# B&R Automation Studio project x20ost
Automation Studio 3.0.71.10

## Configuration Config1

### Task classes (Cpu.sw)
```
Cyclic#4:
  bnrmain <- bnrmain.prg
DataObjects: FlashModul
Binaries: gcloader, iomap, arconfig, asfw, sysconf
Libraries: DataObj, DM_lib, sys_lib, runtime, burtrap, CAN_Lib, AsTCP, dvframe
```

### IoMap.iom - PLC1/IoMap.iom
```iecst
(********************************************************************
 * COPYRIGHT --
 ********************************************************************
 * File: IoMap.iom
 * Author: a2000
 * Created: December 09, 2009
 ********************************************************************
 * IO mapping file
 ********************************************************************)
VAR_CONFIG
	uiValueAI4_0 AT %IW.IF4.ST3.AnalogInput01;
	uiValueAI4_1 AT %IW.IF4.ST3.AnalogInput02;
	uiValueAI5_0 AT %IW.IF4.ST4.Temperature01;
	uiValueAI5_1 AT %IW.IF4.ST4.Temperature02;
	uiValueAO6_0 AT %QW.IF4.ST5.AnalogOutput01;
	uiValueAO6_1 AT %QW.IF4.ST5.AnalogOutput02;
	uiValueAO6_2 AT %QW.IF4.ST5.AnalogOutput03;
	uiValueAO6_3 AT %QW.IF4.ST5.AnalogOutput04;
	blValueDI7_0 AT %IX.IF4.ST6.DigitalInput01;
	blValueDI7_1 AT %IX.IF4.ST6.DigitalInput02;
	blValueDI7_2 AT %IX.IF4.ST6.DigitalInput03;
	blValueDI7_3 AT %IX.IF4.ST6.DigitalInput04;
	blValueDI7_4 AT %IX.IF4.ST6.DigitalInput05;
	blValueDI7_5 AT %IX.IF4.ST6.DigitalInput06;
	blValueDI7_6 AT %IX.IF4.ST6.DigitalInput07;
	blValueDI7_7 AT %IX.IF4.ST6.DigitalInput08;
	blValueDI7_8 AT %IX.IF4.ST6.DigitalInput09;
	blValueDI7_9 AT %IX.IF4.ST6.DigitalInput10;
	blValueDI7_10 AT %IX.IF4.ST6.DigitalInput11;
	blValueDI7_11 AT %IX.IF4.ST6.DigitalInput12;
	blValueDI8_0 AT %IX.IF4.ST7.DigitalInput01;
	blValueDI8_1 AT %IX.IF4.ST7.DigitalInput02;
	blValueDI8_2 AT %IX.IF4.ST7.DigitalInput03;
	blValueDI8_3 AT %IX.IF4.ST7.DigitalInput04;
	blValueDI8_4 AT %IX.IF4.ST7.DigitalInput05;
	blValueDI8_5 AT %IX.IF4.ST7.DigitalInput06;
	blValueDI8_6 AT %IX.IF4.ST7.DigitalInput07;
	blValueDI8_7 AT %IX.IF4.ST7.DigitalInput08;
	blValueDI8_8 AT %IX.IF4.ST7.DigitalInput09;
	blValueDI8_9 AT %IX.IF4.ST7.DigitalInput10;
	blValueDI8_10 AT %IX.IF4.ST7.DigitalInput11;
	blValueDI8_11 AT %IX.IF4.ST7.DigitalInput12;
	blValueDO9_0 AT %QX.IF4.ST8.DigitalOutput01;
	blValueDO9_1 AT %QX.IF4.ST8.DigitalOutput02;
	blValueDO9_2 AT %QX.IF4.ST8.DigitalOutput03;
	blValueDO9_3 AT %QX.IF4.ST8.DigitalOutput04;
	blValueDO9_4 AT %QX.IF4.ST8.DigitalOutput05;
	blValueDO9_5 AT %QX.IF4.ST8.DigitalOutput06;
	blValueDO9_6 AT %QX.IF4.ST8.DigitalOutput07;
	blValueDO9_7 AT %QX.IF4.ST8.DigitalOutput08;
	blValueDO9_8 AT %QX.IF4.ST8.DigitalOutput09;
	blValueDO9_9 AT %QX.IF4.ST8.DigitalOutput10;
	blValueDO9_10 AT %QX.IF4.ST8.DigitalOutput11;
	blValueDO9_11 AT %QX.IF4.ST8.DigitalOutput12;
	blValueDO10_0 AT %QX.IF4.ST9.DigitalOutput01;
	blValueDO10_1 AT %QX.IF4.ST9.DigitalOutput02;
	blValueDO10_2 AT %QX.IF4.ST9.DigitalOutput03;
	blValueDO10_3 AT %QX.IF4.ST9.DigitalOutput04;
	blValueDO10_4 AT %QX.IF4.ST9.DigitalOutput05;
	blValueDO10_5 AT %QX.IF4.ST9.DigitalOutput06;
	blValueDO10_6 AT %QX.IF4.ST9.DigitalOutput07;
	blValueDO10_7 AT %QX.IF4.ST9.DigitalOutput08;
	blValueDO10_8 AT %QX.IF4.ST9.DigitalOutput09;
	blValueDO10_9 AT %QX.IF4.ST9.DigitalOutput10;
	blValueDO10_10 AT %QX.IF4.ST9.DigitalOutput11;
	blValueDO10_11 AT %QX.IF4.ST9.DigitalOutput12;
END_VAR
```

## Logical view

Binary libraries used (declarations not repeated): Convert, Runtime, Operator, DataObj, DM_lib, sys_lib, CAN_Lib, AsTCP, dvframe


### Program Logical/bnrmain (ANSIC) - A new program

#### bnrmain.c - Implementation code
```c
/********************************************************************
 * COPYRIGHT -- Kontora
 ********************************************************************
 * Program: bnrmain
 * File: bnrmain.c
 * Author: Abramenya
 * Created: January 19, 2009
 ********************************************************************
 * Implementation of program bnrmain
 ********************************************************************/
#include "bnrmain.h"
#include "bnrhconfig.h"
#ifdef _DEFAULT_INCLUDES
 #include <AsDefault.h>
#endif
#ifdef WIN32
//size_t szMem;
#endif
_GLOBAL SYSxinfo_typ SYSXInfo0,SYSXInfo1;
_GLOBAL RTCtime_typ RTCGetTime, RTCSetTime;
_GLOBAL BYTE  m_byObsSystemIntState;
_GLOBAL DWORD m_dwTicTime;
CProcManager *m_pProcManager;
_GLOBAL PVOID pProcManager;
_GLOBAL PVOID pSystem;
_GLOBAL PVOID pDebMsg;
_GLOBAL DWORD nMemSize;
_GLOBAL PVOID pvMEM;
typedef struct _tagMem
{
	WORD nSize;
	void *pvMem;
}PMEM;
//_GLOBAL PMEM *m_pMEM;
extern SLMESSAGE *m_pDebMsg;
extern SHARDCOMPUTERTABLE nConfigTable;

void _INIT bnrmainINIT( void )
{
	SYSxinfo(&SYSXInfo0);
	InitSystem();
	SYSxinfo(&SYSXInfo1);
}
//Cyclic Section
_GLOBAL INT nCTT;
void _CYCLIC bnrmainCYCLIC( void )
{
	if(m_pProcManager!=0)
	m_pProcManager->Run(m_pProcManager);
	nCTT++;
	 //RTC_gettime(&RTCGetTime);
}
//Exit Section
void _EXIT bnrmainEXIT( void ){}
void InitSystem(void)
{
    InitHardValue();
    //printf("\nPre Mem");heapdump();

	m_dwTicTime = SYSTEM_QTIME;
	New(sizeof(SLMESSAGE),m_pDebMsg);

	////PMEM **m_pMEM;
	////New(sizeof(PMEM**),m_pMEM);
	////New(300*sizeof(PVOID),pvMEM);
	////pvMEM

	CreateProcManager();
	CreateSystem(&nConfigTable);
	m_pProcManager->Start(m_pProcManager);

	//pProcManager = m_pProcManager;
	//pSystem = m_pSystem;
	//pDebMsg = m_pDebMsg;
	//nMemSize = nMemSize;

	//printf("\n(__)Memory : %d",nMemSize);
	//Info("\n(__)Memory:&",&nMemSize);
	//printf("\nPost Mem");heapdump();
    //DeleteSystem();
	//nMemSize = nMemSize;
	//Status = SYSxinfo(&SYSXInfo2);
	//printf("\nPost Del Mem");heapdump();
}
void DeleteSystem(void)
{
    /*
	m_pProcManager = pProcManager;
	m_pSystem = pSystem;
	m_pDebMsg = pDebMsg;
    m_pProcManager->Stop(m_pProcManager);
	DestroyObject(CSystem,m_pSystem);
	DestroyObject(CProcManager,m_pProcManager);
	Delete(sizeof(SMESSAGE),m_pDebMsg);
	m_pProcManager = 0;
	*/
}

#ifdef WIN32
int main(void)
{
	bnrmainINIT();
	CreateCyclicProc();
	while (1)
	{
	  GetSysCommand();
	  Sleep(100);
	}
    return 0;
}
void GetSysCommand(void)
{
	int ch;
	int i=0;
	SMESSAGE sMsg;
	while((ch = getchar()) != 0x0a)
	{
	 if (i<DEV_MAX_MSG_SIZE)
	 sMsg.m_sbyInfo[1+i] = (BYTE)ch;
	 i++;
	}
	if(i>0)
	{
	 sMsg.m_sbyInfo[0]   = i+1;
     sMsg.m_swLen        = 9+i+1;
	 sMsg.m_sbyFrom      = MDL_ARMMD;
	 sMsg.m_sbyFor       = MDL_HCOMM;
	 sMsg.m_sbyIntType   = DEV_ARM_PORT_TCP;
	 sMsg.m_sbyServerID  = 0;
	 sMsg.m_sbyType      = EV_DEBMS_DEBOUT_IND;
	 sMsg.m_sbyDirection = 0xff;
	 sMsg.m_sbySensor    = 0xff;
	 //Info("\n(##)CMAIN::>HHAND:%m",(BYTE*)&sMsg);
	 FPUT(DEV_ADMIN_BOX_ID,(BYTE*)&sMsg);
	}
}
#endif
BOOL CreateProcManager(void)
{
	m_pProcManager = NULL;
	New(sizeof(CProcManager),m_pProcManager);
	InitObject(CProcManager,m_pProcManager);
	if(m_pProcManager!=NULL)
	{
	 m_pProcManager->Init(m_pProcManager,m_dwTicTime,TRUE);
 	 return TRUE;
	}else return FALSE;

}
BOOL CreateSystem(SHARDCOMPUTERTABLE *plConfigTable)
{
	m_pSystem = NULL;
	New(sizeof(CSystem),m_pSystem);
	InitObject(CSystem,m_pSystem);
	if (m_pSystem!=NULL)
	{
	 m_pSystem->CreateSystem(m_pSystem,plConfigTable);
	 return TRUE;
	}else return FALSE;
}
void DeleteTimer(PVOID pV)
{
    CSystemTimer *p;
	p = (CSystemTimer*)pV;
	m_pProcManager->DisconnectTimer(m_pProcManager,p);
}
void CrateTimer(PVOID pV)
{
    CSystemTimer *p;
	p = (CSystemTimer*)pV;
	m_pProcManager->ConnectTimer(m_pProcManager,p);
}

void CrateProcess(PVOID pV,SINT* chProcName,BYTE byStateProc,BYTE byPeriod)
{
	 CCyclicSystem *p;
	 p = (CCyclicSystem*)pV;
	 p->Create(p,chProcName,byStateProc,byPeriod);
	 m_pProcManager->ConnectProc(m_pProcManager,p);
}
_GLOBAL BYTE nYear;
void GetCurTime(STIME *pTime)
{
    #ifdef WIN32
    SYSTEMTIME nTM; WORD mSec;
	GetLocalTime(&nTM);
	pTime->tYear  = (BYTE)nTM.wYear-2000;
	pTime->tMonth = (BYTE)nTM.wMonth;
	pTime->tDay   = (BYTE)nTM.wDay;
	pTime->tHour  = (BYTE)nTM.wHour;
	pTime->tMin   = (BYTE)nTM.wMinute;

	pTime->tSec   = (BYTE)nTM.wSecond;
	mSec          = nTM.wMilliseconds + nTM.wSecond*1000;
	pTime->tMSecL = (BYTE)mSec;
	pTime->tMSecH = mSec>>8;
    #else
 	/*
      RTCSetTime.year = 2000;
      RTCSetTime.month = RTCGetTime.month;
      RTCSetTime.day = RTCGetTime.day;
      RTCSetTime.hour = RTCGetTime.hour;
      RTCSetTime.minute = RTCGetTime.minute;
      RTCSetTime.second = RTCGetTime.second;
      RTCSetTime.millisec = RTCGetTime.millisec;
      RTCSetTime.microsec = RTCGetTime.microsec;
	*/
    RTC_gettime(&RTCGetTime);
	pTime->tYear  = (RTCGetTime.year-2000);
	nYear = pTime->tYear;
	pTime->tMonth = RTCGetTime.month;
	pTime->tDay   = RTCGetTime.day;
	pTime->tHour  = RTCGetTime.hour;
	pTime->tMin   = RTCGetTime.minute;
	pTime->tSec   = RTCGetTime.second;
	RTCGetTime.millisec = RTCGetTime.millisec + ((UINT)RTCGetTime.second)*1000;
	pTime->tMSecL = (BYTE)RTCGetTime.millisec;
	pTime->tMSecH = (BYTE)(RTCGetTime.millisec>>8);
    #endif
}
void SetBoardTime(BYTE *byTime)
{
	RTCtime_typ RTCSetTime;
	BYTE nSec;
	WORD nMsec;
	RTCSetTime.year     = 2000+byTime[6];
	RTCSetTime.month    = byTime[5];
	RTCSetTime.day      = byTime[4];
	RTCSetTime.hour     = byTime[3];
	RTCSetTime.minute   = byTime[2];

	nMsec = ((WORD)byTime[0])|((WORD)byTime[1])<<8;
	nSec  = nMsec/1000;
    nMsec = nMsec - nSec*1000;

	RTCSetTime.second   = nSec;
	RTCSetTime.millisec = nMsec;
	//Info("\nYR:%w MN:%b DY:%b HR:%b MI:%b SC:%b MS:%w",&RTCSetTime.year,&RTCSetTime.month,&RTCSetTime.day,&RTCSetTime.hour,&RTCSetTime.minute,&nSec,&nMsec);
    #ifndef WIN32
	RTC_settime(&RTCSetTime);
    #endif
}
void SendSMessage(BYTE byBox,BYTE byFor,BYTE byType)
{
    SHORTMESSAGE m_sMsg;
	m_sMsg.m_swLen        = 9;
	m_sMsg.m_sbyFrom      = DIR_PHMDL;
	m_sMsg.m_sbyFor       = byFor;
	m_sMsg.m_sbyIntType   = 0;
	m_sMsg.m_sbyServerID  = 0;
	m_sMsg.m_sbyType      = byType;
	m_sMsg.m_sbyDirection = 0;
	m_sMsg.m_sbySensor    = 0;
	FPUT(byBox,(BYTE*)&m_sMsg);
    #ifdef DEB_CMain
	Info("\n(__)CMAIN::>OUTT::%M",&m_sMsg);
    #endif
}
void SendCommand(BYTE byEvent,SINT *pchCommand)
{
	SHORTMESSAGE m_sMsg;
	BYTE byNbLen;
	m_sMsg.m_sbyFrom      = DIR_KPMOD;
	m_sMsg.m_sbyFor       = DIR_KPTO101;
	m_sMsg.m_sbyIntType   = 0;
	m_sMsg.m_sbyServerID  = 0;
	m_sMsg.m_sbyType      = byEvent;
	m_sMsg.m_sbyDirection = 0;
	m_sMsg.m_sbySensor    = 0;
	byNbLen = strlen(pchCommand);
    memcpy(m_sMsg.m_sbyInfo,pchCommand,byNbLen);
	m_sMsg.m_sbyInfo[byNbLen] = 13;
	m_sMsg.m_sbyInfo[byNbLen+1] = 10;
	m_sMsg.m_swLen            = 9+byNbLen+2;
	#ifdef DEB_CMain
    Info("\n(__)CMAIN::>Command:%s",pchCommand);
    #endif
	FPUT(DEV_RSMMD_BOX_ID,(BYTE*)&m_sMsg);
}
void SendChar(BYTE byEvent,SINT *pchCommand)
{
	SHORTMESSAGE m_sMsg;
	BYTE byNbLen;
	m_sMsg.m_sbyFrom      = DIR_KPMOD;
	m_sMsg.m_sbyFor       = DIR_KPTO101;
	m_sMsg.m_sbyIntType   = 0;
	m_sMsg.m_sbyServerID  = 0;
	m_sMsg.m_sbyType      = byEvent;
	m_sMsg.m_sbyDirection = 0;
	m_sMsg.m_sbySensor    = 0;
	byNbLen = strlen(pchCommand);
    memcpy(m_sMsg.m_sbyInfo,pchCommand,byNbLen);
	//m_sMsg.m_sbyInfo[byNbLen] = 13;
	//m_sMsg.m_sbyInfo[byNbLen+1] = 10;
	m_sMsg.m_swLen            = 9+byNbLen;
	//#ifdef DEB_CMain
    //Info("\n(__)CMAIN::>Command:%s",pchCommand);
    //#endif
	FPUT(DEV_RSMMD_BOX_ID,(BYTE*)&m_sMsg);
}
_GLOBAL INT nQMem;
void NEW(int nSize,void **pVoid)
{
     #ifdef WIN32
	 MEM_alloc(nSize,*pVoid);
     #else
	 MEM_alloc(nSize,pVoid);
     #endif
	 nQMem++;
	 nMemSize += nSize;
};
void FREE(int nSize,void **pVoid)
{
	 if(nSize!=0)
     MEM_free(nSize,pVoid);
	 nMemSize -= nSize;
}
#ifdef WIN32
DWORD WINAPI CyclicProcess( PVOID pVoid)
{
	HANDLE hEvent = CreateEvent(NULL,FALSE,TRUE,NULL);
	int nTime;
	while (1)
	{
	 bnrmainCYCLIC();
	 WaitForSingleObject(hEvent,m_dwTicTime);
	 //if (nTime%50==0) Info("\nTMR_________");
	 //nTime++;
	 //Sleep(20);
	 //Sleep(m_dwTicTime);
	}
	return 0;
}
void CreateCyclicProc(void)
{
	DWORD dwThreadId, dwThrdParam = 1;
	HANDLE hThread;
	hThread = CreateThread(NULL,0,CyclicProcess,&dwThrdParam,0,&dwThreadId);
}
void heapdump( void )
{
	_HEAPINFO hinfo;
	int heapstatus;
	hinfo._pentry = NULL;
	while( ( heapstatus = _heapwalk( &hinfo ) ) == _HEAPOK )
	{ printf( "%6s block at %Fp of size %4.4X\n",
	( hinfo._useflag == _USEDENTRY ? "USED" : "FREE" ),
	hinfo._pentry, hinfo._size );
	}

	switch( heapstatus )
	{
	case _HEAPEMPTY:
		printf( "OK - empty heap\n" );
		break;
	case _HEAPEND:
		printf( "OK - end of heap\n" );
		break;
	case _HEAPBADPTR:
		printf( "ERROR - bad pointer to heap\n" );
		break;
	case _HEAPBADBEGIN:
		printf( "ERROR - bad start of heap\n" );
		break;
	case _HEAPBADNODE:
		printf( "ERROR - bad node in heap\n" );
		break;
	}
}
#endif
```

#### bnradmin.c
```c
/********************************************************************
 * COPYRIGHT -- Kontora
 ********************************************************************
 * Program: bnrmain
 * File: bnrlsens.c
 * Author: Abramenya
 * Created: January 19, 2009
 *******************************************************************/

#include "bnradmin.h"
#include "bnrpob.h"
#ifdef _DEFAULT_INCLUDES
 #include <AsDefault.h>
#endif
#define SYS_REQ_ALL_PARAM                0x6673 // isf - Авария интерфейса
#define SYS_SET_OUT                      0x746f // iot xxx
#define SYS_SET_OUT_BOX                  0x626f // iob xxx
#define SYS_SET_TST_MSG                  0x6d74 // itm xxx
#define SYS_SET_OUT_DIR                  0x736f // iob xxx
#define SYS_SET_DEV_VER                  0x766f // iov xxx
extern SSOFTSWITCHTABLE nSoftSwitchTable;
extern BOOL *blpValueDI8[];
extern UINT *uipValueAI2[];

extern BOOL *blpAlValueAI2[];
extern BOOL *blAsValueAI[];
//_GLOBAL INT iCAdminVal;
SINT *chAdmState[] =
{
	"ST00_NULL",
    "ST01_DISC",
	"ST02_CONN",
	"ST03_WAIT_CONF",
	"ST04_SYST_READY",
	"ST05_WAIT_READY",
};
_GLOBAL INT16 wTICode,nSG;
void CAdmin_Init(This)
{
     DECLARE_MULTI_OPEN(CAdmin,CCyclicSystem)
     #ifdef DEB_CAdmin
	 Info("\n(__)CADMN::>Create Admin.");
     #endif
	 wTICode = 0;
	 nSG     = 0;
	 //pT->m_blArmState = FALSE;
	 //dwFL  |= DEB_OUT_BOX_ADMIN;
	 //dwFL = 48;
	 pB->SetBoxID(pB,DEV_ADMIN_BOX_ID);
	 pT->m_bySystemState = SYS_ST01_DISC;
	 pT->m_blArmState = TRUE;
}
_GLOBAL UINT nTICHA;
void CAdmin_CyclicProc(This)
{
     DECLARE_MULTI_OPEN(CAdmin,CCyclicSystem)
	 pB->m_dwAmoutQuant++;

	 if(wTICode>=32000)
	 nSG = -400;
	 if(wTICode<=0)
	 nSG = 400;

	 //wTICode =  wTICode + nSG;
	 //*uipValueAI2[0] = wTICode;

	 //nTICHA++;
	 //if ((nTICHA % 2)==0)
	 //Info("\n(__)CADMN::>TI:%w",uipValueAI2[0]);
}

void CAdmin_SetSystemID(This,BYTE bySystemID)
{
     DECLARE_MULTI_OPEN(CAdmin,CCyclicSystem)
	 pT->m_bySystemID = bySystemID;
}
BOOL CAdmin_EventHandler(This,SMESSAGE *pMsg)
{
	 BOOL res = TRUE;
     DECLARE_MULTI_OPEN(CAdmin,CCyclicSystem)
	 BYTE byState;
	 byState = pT->GetState(pT);
	 switch (pMsg->m_sbyFor)
	 {
		case MDL_HCOMM:
			 pT->PreCommHandler(pT,pMsg);
		break;
		case MDL_ADMIN:
			 pT->AdminAutomat(pT,pMsg);
		break;
		case MDL_SYSTM:
		break;
		case MDL_DIRMD:
		break;
		case MDL_COMPT:
		break;
		default:
		break;
	 }
	 return res;
}
BOOL CAdmin_AdminAutomat(This,SMESSAGE *pMsg)
{
     DECLARE_MULTI_OPEN(CAdmin,CCyclicSystem)
	 BOOL res = FALSE;
	 BYTE byEvent = pMsg->m_sbyType;
	 switch(pT->GetState(pT))
	 {
	    case SYS_ST00_NULL:
        break;
	    case SYS_ST01_DISC:
			 if((byEvent==EV_ADMIN_ARM_CONN_IND))
			 {
              #ifdef DEB_CAdmin
			  Info("\n(%b)CADMN::>ARM_CONN_IND:%M",&pT->m_bySystemID,(BYTE*)pMsg);
              #endif
			  pT->m_blArmState = TRUE;
              pT->SendMessage(pT,DEV_ARMOT_BOX_ID,MDL_ARMSY,EV_ADMIN_ARM_CONN_IND,0,0);
			  pT->SendMessage(pT,DEV_ARMOT_BOX_ID,MDL_ARMSY,EV_ADMIN_SYS_CONFIG_IND,0,0); //Запросить конфигурацию
			  pT->m_pTAskConfig.OnTimer(&pT->m_pTAskConfig,T4SEC);
			  pT->SetState(pT,SYS_ST03_WAIT_CONF);
			  res = TRUE;
			 }
        break;
		case SYS_ST02_CONN:
        break;
	    case SYS_ST03_WAIT_CONF:
			 if(byEvent==EV_ADMIN_ASK_CONF_TIM_IND)
			 {
              #ifdef DEB_CAdmin
			  Info("\n(%b)CADMN::>ASK_CONF_TIM_IND:%M",&pT->m_bySystemID,(BYTE*)pMsg);
              #endif
			  pT->SendMessage(pT,DEV_ARMOT_BOX_ID,MDL_ARMSY,EV_ADMIN_SYS_CONFIG_IND,0,0); //Запросить конфигурацию
			  pT->m_pTAskConfig.OnTimer(&pT->m_pTAskConfig,T4SEC);
			  res = TRUE;
			 }else
			 if(byEvent==EV_ADMIN_SYS_CONFIG_REQ)
			 {
              #ifdef DEB_CAdmin
			  Info("\n(%b)CADMN::>SYS_CONFIG_REQ:%M",&pT->m_bySystemID,(BYTE*)pMsg);
              #endif
			  pT->m_pTAskConfig.OfTimer(&pT->m_pTAskConfig);
			  pT->SendMessage(pT,DEV_SYSTM_BOX_ID,MDL_SYSTM,EV_SYSTM_INIT_OBS_REQ,0,0);
			  res = TRUE;
			 }else
			 if(byEvent==EV_SYSTM_INIT_OBS_IND)
			 {
              #ifdef DEB_CAdmin
			  Info("\n(%b)CADMN::>INIT_OBS_IND:%M",&pT->m_bySystemID,(BYTE*)pMsg);
              #endif
			  Info("\n(%b)CADMN::>B&R System Ready!",&pT->m_bySystemID);
			  pT->SendMessage(pT,DEV_ARMOT_BOX_ID,MDL_ARMSY,EV_ADMIN_SYS_READY_IND,0,0);
			  pT->SetState(pT,SYS_ST04_SYST_READY);
			  res = TRUE;
			 }
			 if(byEvent==EV_ADMIN_ARM_DISC_IND)pT->SetState(pT,SYS_ST01_DISC);
        break;
		case SYS_ST05_WAIT_READY:
			 switch(byEvent)
			 {
			  case EV_ADMIN_TMR_SSTATE_IND:
				   pT->SendMessage(pT,DEV_ARMOT_BOX_ID,MDL_ARMSY,EV_ADMIN_SYS_READY_IND,0,0);
				   pT->m_pTSendState.OnTimer(&pT->m_pTSendState,T4SEC);
			  break;
			  case EV_ADMIN_ARM_READY_REQ:
				   //pT->m_pTSendState->OfTimer(pT->m_pTSendState);
				   pT->SendMessage(pT,DEV_ARMOT_BOX_ID,MDL_ARMSY,EV_ADMIN_SYS_READY_IND,0,0);
				   pT->m_blArmState = TRUE;
				   pT->SetState(pT,SYS_ST04_SYST_READY);
			  break;
			  default:
			  break;
			 }
		break;
	    case SYS_ST04_SYST_READY:
			 switch(byEvent)
			 {
			  case EV_ADMIN_ARM_READY_REQ:
				   pT->SendMessage(pT,DEV_ARMOT_BOX_ID,MDL_ARMSY,EV_ADMIN_SYS_READY_IND,0,0);
			  break;
			  case EV_ADMIN_ARM_DISC_IND:
				   //pT->m_pTSendState->OnTimer(pT->m_pTSendState,T4SEC);
				   pT->SetState(pT,SYS_ST05_WAIT_READY);
				   pT->m_blArmState = FALSE;
			  break;
			  case EV_ADMIN_SET_ALM_HILEV_REQ: //Авария превышения верхнего ав. предела 	68
                   #ifdef DEB_CAdmin
			       Info("\n(%b)CADMN::>SET_ALM_HILEV_REQ:%M",&pT->m_bySystemID,(BYTE*)pMsg);
                   #endif
			   	   pT->SendMessage(pT,DEV_ARMOT_BOX_ID,MDL_ARMSY,pMsg->m_sbyType,pMsg->m_sbyDirection,pMsg->m_sbySensor);
			  break;
			  case EV_ADMIN_REM_ALM_HILEV_REQ: //Устранение аварии превышения верхнего ав. предела 	69
                   #ifdef DEB_CAdmin
			       Info("\n(%b)CADMN::>REM_ALM_HILEV_REQ:%M",&pT->m_bySystemID,(BYTE*)pMsg);
                   #endif
			       pT->SendMessage(pT,DEV_ARMOT_BOX_ID,MDL_ARMSY,pMsg->m_sbyType,pMsg->m_sbyDirection,pMsg->m_sbySensor);
			  break;
			  case EV_ADMIN_SET_ALM_LOLEV_REQ: //Авария превышения нижнего ав. предела 	70
                   #ifdef DEB_CAdmin
			       Info("\n(%b)CADMN::>REM_ALM_LOLEV_REQ:%M",&pT->m_bySystemID,(BYTE*)pMsg);
                   #endif
			       pT->SendMessage(pT,DEV_ARMOT_BOX_ID,MDL_ARMSY,pMsg->m_sbyType,pMsg->m_sbyDirection,pMsg->m_sbySensor);
			  break;
			  case EV_ADMIN_REM_ALM_LOLEV_REQ: //Устранение аварии превышения нижнего ав. предела 	71
                   #ifdef DEB_CAdmin
			       Info("\n(%b)CADMN::>REM_ALM_LOLEV_REQ:%M",&pT->m_bySystemID,(BYTE*)pMsg);
                   #endif
			       pT->SendMessage(pT,DEV_ARMOT_BOX_ID,MDL_ARMSY,pMsg->m_sbyType,pMsg->m_sbyDirection,pMsg->m_sbySensor);
			  break;
	          case EV_ADMIN_ARM_STOP_REQ:
		           //pT->CloseInterface(pC);
			       //Info("\n(%b)CADMN::>EV_ADMIN_ARM_STOP_REQ:%M",&pT->m_bySystemID,(BYTE*)pMsg);
	       	  break;
			 }
        default:
		break;
	 }
	 return res;
}
BOOL CAdmin_SendMessage(This,BYTE byBox,BYTE byFor,BYTE byType,BYTE byDir,BYTE bySens)
{
     DECLARE_MULTI_OPEN(CAdmin,CCyclicSystem)
	 BOOL res = TRUE;
	 SHORTMESSAGE m_sMsg;
	 m_sMsg.m_swLen        = 9;
	 m_sMsg.m_sbyFrom      = MDL_ADMIN;
	 m_sMsg.m_sbyFor       = byFor;
	 m_sMsg.m_sbyIntType   = DEV_SYS_INTERFACE;
	 m_sMsg.m_sbyServerID  = pT->m_bySystemID;
	 m_sMsg.m_sbyType      = byType;
	 m_sMsg.m_sbyDirection = byDir;
	 m_sMsg.m_sbySensor    = bySens;
	 //if(pT->m_blArmState)
     FPUT(byBox,(BYTE*)&m_sMsg);
	 return res;
}
void CAdmin_PreCommHandler(This,SMESSAGE *pMsg)
{
     DECLARE_MULTI_OPEN(CAdmin,CCyclicSystem)
	 BYTE byLength;
	 DWORD Code;
	 BYTE ps,*pD=(BYTE*)&Code;
     #ifdef DEB_CAdmin
 	 Info("\n(__)CHAND::>HSYST_O <- %m",pMsg->m_sbyInfo);
     #endif
	 Code = 0;
	 byLength = pMsg->m_sbyInfo[0];
	 for (ps = 0;ps<byLength;ps++)
	 if ((char)pMsg->m_sbyInfo[ps]==' ')
	 break;
	 if (ps<=MAX_COMMAND_LENGTH)
	 {
	 #ifdef WIN32
	 memcpy(&Code,&pMsg->m_sbyInfo[2],ps-2);
	 #else
	 pD[3] = pMsg->m_sbyInfo[2];
	 pD[2] = pMsg->m_sbyInfo[3];
	 #endif
	 pT->HandCommHandler(pT,Code,ps,pMsg->m_sbyInfo,byLength);

	 }
}
void CAdmin_HandCommHandler(This,DWORD b_lCode,BYTE ps,BYTE *pbyBuffer,BYTE byLength)
{
     DECLARE_MULTI_OPEN(CAdmin,CCyclicSystem)
	 SHORTMESSAGE m_sMsg;
	 BYTE byParam0,byParam1;
	 WORD wValue;
	 #ifdef DEB_CAdmin
	 //Info("\n(##)CHAND::>Code:%d, PS:%b LN:%b MS0:%b",&b_lCode,&ps,&byLength,&pbyBuffer[ps]);
     #endif
	 switch(b_lCode)
	 {
       case SYS_REQ_ALL_PARAM:
		   if (ps<(byLength-1))
		   {
            ps++;
			byParam0=pbyBuffer[ps]-0x30;
		    //Info("\nCHAND::>Command SYS_REQ_ALL_PARAM.Param0:%b",&byParam0);
		   }
	   break;
       case SYS_SET_TST_MSG:// itm xxx
		    if (ps<(byLength-1))
			{
			   ps++;
			   byParam0=pbyBuffer[ps]-0x30;
			   ps++;
			   byParam1=pbyBuffer[ps]-0x30;
               #ifdef DEB_CAdmin
			   Info("\n(__)CHAND::>SET DIG PIN[%b]:STT[%b]",&byParam0,&byParam1);
			   #endif
			   *blpValueDI8[byParam0] = byParam1;
			   //*blpAlValueAI2[byParam0] = byParam1;
			   //*blAsValueAI = byParam1;
			   //Info("\n(%b)SetPin In %b",&byParam0,&byParam1);
			}
	   break;
       case SYS_SET_OUT://iot
		   {
		    ps++;
		    if((pbyBuffer[ps]-0x30)) dwFL |= DEB_OUT_CYC_ADMIN;else dwFL &= ~DEB_OUT_CYC_ADMIN;
		    ps++;
		    if((pbyBuffer[ps]-0x30)) dwFL |= DEB_OUT_CYC_SYSTM;else dwFL &= ~DEB_OUT_CYC_SYSTM;
		    ps++;
		    if((pbyBuffer[ps]-0x30)) dwFL |= DEB_OUT_CYC_OBSRV;else dwFL &= ~DEB_OUT_CYC_OBSRV;
			ps++;
			if((pbyBuffer[ps]-0x30)) dwFL |= DEB_OUT_PMAN_STAT;else dwFL &= ~DEB_OUT_PMAN_STAT;
		    Info("\n(__)CHAND::>Out SYS_SET_OUT[%w] ",&dwFL);
		   }
       break;
       case SYS_SET_OUT_DIR://ios
		   {
		    ps++;
		    if((pbyBuffer[ps]-0x30)) dwFL |= DEB_OUT_OBSR_COMM;else dwFL &= ~DEB_OUT_OBSR_COMM;
		    ps++;
		    if((pbyBuffer[ps]-0x30)) dwFL |= DEB_OUT_DIRC_COMM;else dwFL &= ~DEB_OUT_DIRC_COMM;
		    Info("\n(__)CHAND::>Out SYS_SET_OUT_DIR[%w] ",&dwFL);
		   }
       break;
	   case SYS_SET_OUT_BOX: //iob
		   {
			ps++;
			if((pbyBuffer[ps]-0x30)) dwFL |= DEB_OUT_BOX_ADMIN;else dwFL &= ~DEB_OUT_BOX_ADMIN;
			ps++;
			if((pbyBuffer[ps]-0x30)) dwFL |= DEB_OUT_BOX_SYSTM;else dwFL &= ~DEB_OUT_BOX_SYSTM;
			ps++;
			if((pbyBuffer[ps]-0x30)) dwFL |= DEB_OUT_BOX_OBSRV;else dwFL &= ~DEB_OUT_BOX_OBSRV;
			Info("\n(__)CHAND::>Out SYS_SET_OUT_[%w]",&dwFL);
		   }
	   break;
	   case SYS_SET_DEV_VER:// iov
           pT->DevVersion(pT) ;
	   break;
	   default:
	   break;
	 };
}
void CAdmin_DevVersion(This)
{
	  DECLARE_MULTI_OPEN(CAdmin,CCyclicSystem)
	  Info("\n/----------------/Automation 2k/---------------------------/");
	  Info("\n/ Объект     :Бобруйский ЗСКГШ............................./");
      #if MYSYSTEM_ID==0
	  Info("\n/ Назначение :Управление параметрами в контуре АС-1......../");
      #elif MYSYSTEM_ID == 1
	  Info("\n/ Назначение :Управление параметрами в контуре АС-2......../");
	  #elif MYSYSTEM_ID == 2
	  Info("\n/ Назначение :Управление параметрами в контуре АС-3......../");
      #elif MYSYSTEM_ID == 3
	  Info("\n/ Назначение :Управление параметрами в контуре КОП........./");
      #elif MYSYSTEM_ID == 4
	  Info("\n/ Назначение :Управление ЧРЭП............................../");
	  #endif
	  Info("\n/ Версия     :[09.09.2009]................................./");
	  Info("\n/ Устройство :Контроллер B&R 2005........................../");
	  Info("\n/ Разработчик:Абраменя Александр Васильевич(2009г)........./");
	  Info("\n/ Тел/mail   :(8-029-563-76-78/alex_mpowt@tut.by)........../");
	  Info("\n/----------------------------------------------------------/");
}
void CAdmin_SetState(This,BYTE byState)
{
     DECLARE_MULTI_OPEN(CAdmin,CCyclicSystem)
     #ifdef DEB_CAdmin
	 Info("\n(%b)CADMN::>State:(%s)->(%s):",&pT->m_bySystemID,chAdmState[pT->m_bySystemState],chAdmState[byState]);
     #endif
     pT->m_bySystemState = byState;
}
BYTE CAdmin_GetState(This)
{
     DECLARE_MULTI_OPEN(CAdmin,CCyclicSystem)
	 return pT->m_bySystemState;
}
void CAdmin_CAdmin(This)
{
     DECLARE_MULTI_OPEN(CAdmin,CCyclicSystem)
	 DECLARE_REGISTRATION(CAdmin,Init)
	 DECLARE_REGISTRATION(CAdmin,SendMessage)
	 DECLARE_REGISTRATION(CAdmin,HandCommHandler)
	 DECLARE_REGISTRATION(CAdmin,PreCommHandler)
	 DECLARE_REGISTRATION(CAdmin,SetSystemID)
	 DECLARE_REGISTRATION(CAdmin,SetState)
	 DECLARE_REGISTRATION(CAdmin,GetState)
	 DECLARE_REGISTRATION(CAdmin,AdminAutomat)
	 DECLARE_REGISTRATION(CAdmin,DevVersion)
	 DECLARE_VIRTUAL_FUNC(CAdmin,CyclicProc)
	 DECLARE_VIRTUAL_FUNC(CAdmin,EventHandler)
	 InitObject(CMTimer,&pT->m_pTAskConfig);
     pT->m_pTAskConfig.SetTimer(&pT->m_pTAskConfig,MDL_ADMIN,MDL_ADMIN,EV_ADMIN_ASK_CONF_TIM_IND,0,0,DEV_ADMIN_BOX_ID);
	 InitObject(CMTimer,&pT->m_pTSendState);
     pT->m_pTSendState.SetTimer(&pT->m_pTSendState,MDL_ADMIN,MDL_ADMIN,EV_ADMIN_TMR_SSTATE_IND,0,0,DEV_ADMIN_BOX_ID);
}
void CAdmin_DCAdmin(This)
{
	 DECLARE_MULTI_OPEN(CAdmin,CCyclicSystem)
}
DECLARE_MULTI_CREATE(CAdmin,CCyclicSystem)
```

#### bnrkp.c
```c
/********************************************************************
 * COPYRIGHT -- Kontora
 ********************************************************************
 * Program: bnrmain
 * File: bnrlsens.c
 * Author: Abramenya
 * Created: January 19, 2009
 *******************************************************************/

#include "bnrkp.h"
#include "bnrmain.h"
#ifdef _DEFAULT_INCLUDES
 #include <AsDefault.h>
#endif
extern SKPPARAM nKP;
extern SARMINTERFACE nARM0;
extern STIPARAMS nTI;
extern STSPARAMS nTS;
extern STUPARAMS nTU;
extern char *STTS[];
_GLOBAL INT nSendTmrQry;
void CKpModule_Init(This,SHARDCOMPUTERTABLE *pPCTable,SSOFTSWITCHTABLE *pKPTable)
{
    DECLARE_MULTI_OPEN(CKpModule,CCyclicSystem)
	BOOL blSerialize;
	//pT->m_byKpID = pKPTable->sDirectionTable[0].byDirectionID;
	FDEFINE(DEV_KPMDL_BOX_ID,DEV_KPMDL_BOX_SZ);
    FDEFINE(BOX_L4,BOX_L4_SZ);
	FDEFINE(BOX_L4_1,BOX_L4_1_SZ);
	nSendTmrQry = 0;
    InitObject(CMFlash,&pT->m_nFlash);
	pT->m_pFlash = &pT->m_nFlash;
    pB->SetBoxID(pB,DEV_KPMDL_BOX_ID);
	pT->m_pPCT   = pPCTable;
	pT->m_pPST   = pKPTable;
	pT->m_pKP    = pPCTable->pKpParam;
	pT->m_byKpID = pT->m_pKP->byKpID;
	pT->m_pD     = &pT->m_pPST->sDirectionTable[0];
	pT->m_wCallTime = pT->m_pKP->byCallPeriod*10;
	pT->m_blDiscStart = FALSE;
	pT->m_byDiscProc  = 0;

	pT->m_byObsObject = 0;
	pT->m_byObsTime   = 0;
	pT->m_blIfConnect = TRUE;

    pT->m_byKpState    = MKP_NULL_ST00;
	//pT->m_byConnCT = 0;
	pT->m_blBufferST = TRUE;
	InitObject(CMTimer,&pT->m_nConnTMR);
	pT->m_nConnTMR.SetTimer(&pT->m_nConnTMR,DIR_KPTOKP,DIR_KPTOKP,EV_TMR_SRR_REQ,0,0,DEV_KPMDL_BOX_ID);

	InitObject(CMTimer,&pT->m_nRepConnTMR);
	pT->m_nRepConnTMR.SetTimer(&pT->m_nRepConnTMR,DIR_KPTOKP,DIR_KPTOKP,EV_TMR_RCAL_REQ,0,0,DEV_KPMDL_BOX_ID);

	InitObject(CMTimer,&pT->m_nDiscTMR);
	pT->m_nDiscTMR.SetTimer(&pT->m_nDiscTMR,DIR_KPTOKP,DIR_KPTOKP,EV_TMR_DISC_REQ,0,0,DEV_KPMDL_BOX_ID);

	InitObject(CMTimer,&pT->m_pResetTimer);
 	pT->m_pResetTimer.SetTimer(&pT->m_pResetTimer,DIR_KPTOKP,DIR_KPTOKP,EV_SYSTM_RESET_TIM_BRD_IND,0,0,DEV_KPMDL_BOX_ID);

	InitObject(CMTimer,&pT->m_nConnRepTMP);
	pT->m_nConnRepTMP.SetTimer(&pT->m_nConnRepTMP,DIR_KPTOKP,DIR_KPTOKP,EV_TMR_CNRP_REQ,0,0,DEV_KPMDL_BOX_ID);

	InitObject(CMTimer,&pT->m_nPuCommTMR);
	pT->m_nPuCommTMR.SetTimer(&pT->m_nPuCommTMR,DIR_KPTOKP,DIR_KPTOKP,EV_TMR_PUCM_REQ,0,0,DEV_KPMDL_BOX_ID);

	InitObject(CMTimer,&pT->m_nSDiscTMR);
	pT->m_nSDiscTMR.SetTimer(&pT->m_nSDiscTMR,DIR_KPTOKP,DIR_KPTOKP,EV_TMR_SDIS_REQ,0,0,DEV_KPMDL_BOX_ID);

	blSerialize = pT->Serialize(pT,FALSE);
	pT->CreateChannels(pT,&pKPTable->sDirectionTable[0]);

	#ifdef DEB_CKpModule
 	Info("\n(__)CKPMD::>Create Kp Module");
    #endif
	//pT->SaveInPin(pT);
}
_GLOBAL BYTE nTUU;
void CKpModule_CreateChannels(This,SDIRTABLE *pDTable)
{
    DECLARE_MULTI_OPEN(CKpModule,CCyclicSystem)
	WORD i;
	CTeleInd *pTI;
	CTeleSignal *pTS;
	CTeleControl *pTU;
	STSPARAM *pPV;
	pT->m_wAmChannel = pDTable->byAmSwitching;
	New(sizeof(CTeleSensor*)*pT->m_wAmChannel,pT->m_pTeleSensor);
	for(i=0;i<pT->m_wAmChannel;i++)
	{
	 pPV = (STSPARAM*)pDTable->pSwitchTable[i];//Find Type
	 switch (pPV->byType)
	 {
	   case TI:
		    New(sizeof(CTeleInd),pTI);
			InitObject(CTeleInd,pTI);
			pTI->pBase->m_pComputer = pT->m_pComputer;
			pT->m_pTeleSensor[i]    = pTI->pBase;
			pTI->pBase->m_pPCT      = pT->m_pPCT;
			pTI->pBase->Init(pTI->pBase,(PVOID)pPV);
	   break;
	   case TS:
		    New(sizeof(CTeleSignal),pTS);
			InitObject(CTeleSignal,pTS);
			pTS->pBase->m_pComputer = pT->m_pComputer;
		    pT->m_pTeleSensor[i]    = pTS->pBase;
			pTS->pBase->m_pPCT      = pT->m_pPCT;
			pTS->pBase->Init(pTS->pBase,(PVOID)pPV);
	   break;
	   case TU:
		    New(sizeof(CTeleControl),pTU);
			InitObject(CTeleControl,pTU);
			pTU->pBase->m_pComputer = pT->m_pComputer;
		    pT->m_pTeleSensor[i]    = pTU->pBase;
			pTU->pBase->m_pPCT      = pT->m_pPCT;
			pTU->pBase->Init(pTU->pBase,(PVOID)pPV);
	   break;
	   default:
	   break;
	 }
	}
}
/*
REG_KPPAR_ADDR=0,
REG_PORTT_ADDR,
REG_HARDT_ADDR,
REG_SOFTI_ADDR,
REG_SOFTS_ADDR,
REG_SOFTU_ADDR,
REG_SOFTR_ADDR,
*/
BOOL CKpModule_EventHandler(This,SMESSAGE *pMsg)
{
    DECLARE_MULTI_OPEN(CKpModule,CCyclicSystem)
	CTeleSensor *pTS;
	WORD wValue = 0;
	BYTE byID;
	BYTE byA0   = pMsg->m_sbyInfo[1];
	BYTE byA1   = pMsg->m_sbyInfo[2];
	BYTE byA2   = pMsg->m_sbyInfo[3];
	BYTE byLen  = pMsg->m_sbyInfo[0];
	WORD wParam;
	#ifdef DEB_CKpModule
	Info("\n(__)CKPMM::>INPT::%M",pMsg);
	#endif
	switch(pMsg->m_sbyFor)
	{
	  case DIR_101TOKP:
		   switch(pMsg->m_sbyType)
		   {
		    case PL_DATA_IND:
				 switch(byA0)
				 {
				   case REG_KPPAR_ADDR:
					    if ((byA1 == CKP_SETT_TIME)||(byA1 == CKP_SETT_KPID))
						{
						    if (byA1 == CKP_SETT_TIME) SetBoardTime(&pMsg->m_sbyInfo[4]);
							pT->m_nPuCommTMR.OfTimer(&pT->m_nPuCommTMR);
							pT->m_nConnTMR.OfTimer(&pT->m_nConnTMR);
							pT->m_nConnRepTMP.OfTimer(&pT->m_nConnRepTMP);
							//pT->m_nRepConnTMR.OfTimer(&pT->m_nRepConnTMR);
							//pT->m_blIfConnect = FALSE;
							#ifdef DEB_CKpModule
	    					Info("\n(__)CKPMM::>PU TIMER OFF");
							#endif
						}
				   	    if (byA1 == CKP_CLSE_PORT) SendSMessage(DEV_RSMMD_BOX_ID,DIR_KPTOPH,PH_CLOSE_PORT_REQ);
						if (byA1 == CKP_SAVE_SETT) {pT->m_nCT.byDefSett = 0;pT->Serialize(pT,TRUE);}
						if (byA1 == CKP_REST_BORD) pT->m_pResetTimer.OnTimer(&pT->m_pResetTimer,100);
						if (byA1 == CKP_REST_12BR)
						{
						 memcpy(&wParam,&pMsg->m_sbyInfo[5],2);
						 pT->m_nCT.byDefSett = (BYTE)wParam;
				         pT->Serialize(pT,TRUE);
						 pT->m_pResetTimer.OnTimer(&pT->m_pResetTimer,100);
						}
						if (byA1 == CKP_STOP_REST) pT->m_pResetTimer.OfTimer(&pT->m_pResetTimer);
						if (byA1 == CKP_FREE_BXL4) FFREE(BOX_L4);
						if (byA1 == CKP_SETT_BL41) pT->SaveInPin(pT);
						if (byA1 == CKP_REMT_DISC) pT->m_nSDiscTMR.OnTimer(&pT->m_nSDiscTMR,30);
						if (byA1 == CKP_SVAL_PINS) pT->SaveAlarmPin(pT);
						if (byA1 == CKP_SVAL_SLOT) pT->SaveSlotState(pT);
						if (byA1 == CKP_STRT_CHTM)
						{
							#ifdef WIN32
							pT->m_byObsObject = pMsg->m_sbyInfo[5];
							pT->m_byObsTime   = pMsg->m_sbyInfo[6]*10;
							#else
							pT->m_byObsObject = pMsg->m_sbyInfo[6];
							pT->m_byObsTime   = pMsg->m_sbyInfo[5]*10;
							#endif
							pT->StartCheck(pT,pT->m_byObsTime,pT->m_byObsObject);
						}
						if (byA1 == CKP_STOP_CHTM) pT->StopCheck(pT);
						if (byA1 == CKP_INIT_PORT) SendSMessage(DEV_RSMMD_BOX_ID,DIR_KPTOPH,PH_INIT_PORT_REQ);

				   break;
				   case REG_PORTT_ADDR:
				   break;
				   case REG_HARDT_ADDR:
				   break;
				   case REG_SOFTI_ADDR:
					    byID = byA1;
						if(byA1<pT->m_pD->byAmTI)
						{
					   	 pTS = pT->m_pTeleSensor[byID];
						 if((byA2==3)||(byA2==4)) pTS->Switch(pTS);
						 pTS->EventHandler(pTS->pChld,pMsg);
						}
				   break;
				   case REG_SOFTS_ADDR:
					    byID = byA1+pT->m_pD->byAmTI;
						if(byA1<pT->m_pD->byAmTS)
						{
					     pTS = pT->m_pTeleSensor[byID];
						 if((byA2==3)||(byA2==4)) pTS->Switch(pTS);
					     pTS->EventHandler(pTS->pChld,pMsg);
						}
				   break;
				   case REG_SOFTU_ADDR:
					    byID = byA1+pT->m_pD->byAmTI+pT->m_pD->byAmTS;
						if(byA1<pT->m_pD->byAmTU)
						{
					     pTS = pT->m_pTeleSensor[byID];
						 if((byA2==3)||(byA2==4)) pTS->Switch(pTS);
					     pTS->EventHandler(pTS->pChld,pMsg);
						}
				   break;
				   case REG_SOFTR_ADDR:
				   break;
				 }
		    break;
			case PH_CONN_IND:
                 #ifdef DEB_CKpModule
				 Info("\n(__)CKPMM::>CONNECT");
                 #endif
				 pT->m_byKpState = MKP_CONN_ST01;
				 pT->m_nPuCommTMR.OnTimer(&pT->m_nPuCommTMR,100);
				 pT->m_nConnTMR.OfTimer(&pT->m_nConnTMR);
				 pT->m_blIfConnect = TRUE;
				 //pT->m_nConnRepTMP.OfTimer(&pT->m_nConnRepTMP);
	             //pT->m_wCallTime = 300;
				 //pT->m_byConnCT  = 0;
				 pT->SaveInPin(pT);
                 //pT->SaveAlarmPin(pT);
				 //pT->SaveSlotState(pT);
			break;
			case PH_DISC_IND:
                 #ifdef DEB_CKpModule
				 Info("\n(__)CKPMM::>DISCONNECT");
                 #endif
				 pT->m_byKpState = MKP_DISC_ST02;
				 pT->m_nDiscTMR.OfTimer(&pT->m_nDiscTMR);
				 pT->m_nConnTMR.OfTimer(&pT->m_nConnTMR);
				 //pT->m_nRepConnTMR.OfTimer(&pT->m_nRepConnTMR);
				 if(FCHECK(BOX_L4)!=0) pT->StartConnect(pT);
				 //pT->m_nConnRepTMP.OfTimer(&pT->m_nConnRepTMP);
	             //pT->m_wCallTime = 600;
				 //pT->m_byConnCT  = 0;
			break;
			default:
            break;
		   }
      break;
	  case DIR_KPTOKP:
		   if (pMsg->m_sbyType==EV_SYSTM_RESET_TIM_BRD_IND)
		   {
            #ifndef WIN32
			SYSreset(1, 2);
            #endif
			pMsg->m_sbyType=EV_SYSTM_RESET_TIM_BRD_IND;
		   }

           if (pMsg->m_sbyType==EV_TMR_SDIS_REQ)
		   {
		   	#ifdef DEB_CKpModule
	        Info("\n(__)CKPMM::>GO REM DISC.");
			#endif
	        pT->Disconnect(pT);
		   }

           if (pMsg->m_sbyType==EV_TMR_PUCM_REQ)
		   {
		   	#ifdef DEB_CKpModule
			Info("\n(__)CKPMM::>PU TIMER EMPTY + DISC.");
			#endif
			pT->m_nConnTMR.OfTimer(&pT->m_nConnTMR);
            pT->Disconnect(pT);
		   }

		   if (pMsg->m_sbyType==EV_TMR_CNRP_REQ)
		   {
		   	#ifdef DEB_CKpModule
		    Info("\n(__)CKPMM::>EV_TMR_CNRP_REQ.");
			#endif
			pT->SendObserveMsg(pT);
		    //pT->StartConnect(pT);
		   }

	       if (pMsg->m_sbyType==EV_TMR_SRR_REQ)
		   {
		   	#ifdef DEB_CKpModule
			Info("\n(__)CKPMM::>EV_TMR_SRR_REQ.");
			#endif
			pT->StartConnect(pT);
		   }

		   if (pMsg->m_sbyType==EV_TMR_RCAL_REQ)
		   {
		   	/*
			#ifdef DEB_CKpModule
			Info("\n(__)CKPMM::>EV_TMR_RCAL_REQ.");
			#endif
			 if((pT->m_byKpState==MKP_DISC_ST02)||(pT->m_byKpState==MKP_NULL_ST00)) pT->StartConnect(pT);
			 else
			 {
			  pT->m_byConnCT  = 0;
		      pT->m_byCallCT  = 3*pT->m_pKP->byAmCall;
			  pT->m_wCallTime = pT->m_pKP->byCallPeriod*10;
			  pT->m_nRepConnTMR.OnTimer(&pT->m_nRepConnTMR,pT->m_wCallTime);
			 }
			 */
		   }

	       if (pMsg->m_sbyType==EV_TMR_DISC_REQ)
		   {
		   	#ifdef DEB_CKpModule
			Info("\n(__)CKPMM::>EV_TMR_DISC_REQ.");
			#endif
			SendCommand(PH_DISC_REQ,"ATH");
			pT->m_byKpState = MKP_NULL_ST00;
			pT->DisconnectL2(pT);
			pT->m_nConnTMR.OnTimer(&pT->m_nConnTMR,30);
			//pT->m_nConnTMR.OnTimer(&pT->m_nConnTMR,pT->m_wCallTime);
		   }
	  break;
	  case DIR_PHTOKP:
	       if (pMsg->m_sbyType==PH_CALL_REQ)
		   {
            #ifdef DEB_CKpModule
			Info("\n(__)CKPMM::>Set Call Proc.");
            #endif
			pT->m_byConnCT  = 0;
		    pT->m_byCallCT  = 3*pT->m_pKP->byAmCall;
			pT->m_wCallTime = pT->m_pKP->byCallPeriod*10;
		    pT->StartConnect(pT);
			//pT->m_wCallTime = pT->m_pKP->byCallPeriod*10;
			//pT->m_nRepConnTMR.OnTimer(&pT->m_nRepConnTMR,pT->m_wCallTime);
		   }
	  break;
	  default:
	  break;
	}
	return TRUE;
}
_GLOBAL INT nSendTmr;
/*
BYTE byAmCall;
BYTE byCallPeriod;
*/
void CKpModule_StartConnect(This)
{
    DECLARE_MULTI_OPEN(CKpModule,CCyclicSystem)
	WORD wTIME = pT->m_pKP->byCallPeriod*10;
	#ifdef DEB_CKpModule
    Info("\n(__)CKPMM::>Start CONNECT::>%b",&pT->m_byConnCT);
    #endif
	if(pT->m_byCallCT--!=0)
	{
     if((pT->m_byKpState==MKP_DISC_ST02)||(pT->m_byKpState==MKP_NULL_ST00))
	 {
	  if(pT->m_byConnCT==0)if(pT->m_pKP->byPhone0[0]!='0'){pT->Connect(pT,pT->m_pKP->byPhone0);wTIME=pT->m_wCallTime;}else wTIME = 10;
	  if(pT->m_byConnCT==1)if(pT->m_pKP->byPhone1[0]!='0'){pT->Connect(pT,pT->m_pKP->byPhone1);wTIME=pT->m_wCallTime;}else wTIME = 10;
	  if(pT->m_byConnCT==2)if(pT->m_pKP->byPhone2[0]!='0'){pT->Connect(pT,pT->m_pKP->byPhone2);wTIME=pT->m_wCallTime;}else wTIME = 10;
	  pT->m_nConnTMR.OnTimer(&pT->m_nConnTMR,wTIME);
	  if(++pT->m_byConnCT>2)pT->m_byConnCT = 0;
	 }else
	 {
      #ifdef DEB_CKpModule
	  Info("\n(__)CKPMM::>Already In Join.Reset Call Proc.");
      #endif
	  pT->m_byCallCT = 3*pT->m_pKP->byAmCall;
	  pT->m_wCallTime = pT->m_pKP->byCallPeriod*10;
	  pT->m_nConnTMR.OnTimer(&pT->m_nConnTMR,pT->m_wCallTime);
	 }
	}else
	{
      #ifdef DEB_CKpModule
	  Info("\n(__)CKPMM::>Join Is Not Installed::%w.",&pT->m_wCallTime);
      #endif
	  pT->m_byCallCT = 3*pT->m_pKP->byAmCall;
	  if (pT->m_blIfConnect==TRUE)
	  {
	   if (pT->m_wCallTime<36000)
	   {
	    pT->m_wCallTime *= 2;
	   }else pT->m_wCallTime = 36000;
	   pT->m_byKpState = MKP_NULL_ST00;
	   pT->m_nConnTMR.OnTimer(&pT->m_nConnTMR,pT->m_wCallTime);
	   pT->m_blIfConnect = FALSE;
	  }else
	  {
	   //pT->m_byCallCT = 3*pT->m_pKP->byAmCall;
	   //pT->m_wCallTime = pT->m_1pKP->byCallPeriod*10;
	   pT->m_blIfConnect = TRUE;
       pT->m_nConnTMR.OnTimer(&pT->m_nConnTMR,60*10);
	  }
	}
}
void CKpModule_Connect(This,SINT *pchPhone)
{
    DECLARE_MULTI_OPEN(CKpModule,CCyclicSystem)
	SINT chPhone[30];
	memset(chPhone,0,sizeof(chPhone));
	strcat(chPhone,"ATD");
    strcat(chPhone,pchPhone);
    SendCommand(PH_CONN_REQ,chPhone);
	/*
	SHORTMESSAGE m_sMsg;
	BYTE byNbLen;
    #ifdef DEB_CKpModule
	Info("\n(__)CKPMM::>Connect Phone:%s",pchPhone);
    #endif
	//SINT *pchPhone;
	m_sMsg.m_sbyFrom      = DIR_KPMOD;
	m_sMsg.m_sbyFor       = DIR_KPTO101;
	m_sMsg.m_sbyIntType   = 0;
	m_sMsg.m_sbyServerID  = 0;
	m_sMsg.m_sbyType      = PH_CONN_REQ;
	m_sMsg.m_sbyDirection = 0;
	m_sMsg.m_sbySensor    = 0;
	m_sMsg.m_sbyInfo[0]   = 'A';
	m_sMsg.m_sbyInfo[1]   = 'T';
	m_sMsg.m_sbyInfo[2]   = 'D';
	byNbLen = strlen(pchPhone);
    memcpy(&m_sMsg.m_sbyInfo[3],pchPhone,byNbLen);
	m_sMsg.m_sbyInfo[2+byNbLen+1] = 13;
	m_sMsg.m_sbyInfo[2+byNbLen+2] = 10;
	m_sMsg.m_swLen                = 9+byNbLen+5;
	//#ifdef DEB_C101Module
    Info("\n(__)CKPMM::>Connect Phone:%s",pchPhone);
    //#endif
	FPUT(DEV_RSMMD_BOX_ID,(BYTE*)&m_sMsg);
	*/

}
void CKpModule_DisconnectL2(This)
{
    DECLARE_MULTI_OPEN(CComServer,CCyclicSystem)
	SHORTMESSAGE m_sMsg;
	m_sMsg.m_swLen        = 9;
	m_sMsg.m_sbyFrom      = DIR_PHMDL;
	m_sMsg.m_sbyFor       = DIR_KPTO101;
	m_sMsg.m_sbyIntType   = 0;
	m_sMsg.m_sbyServerID  = 0;
	m_sMsg.m_sbyType      = PH_DISC_IND;
	m_sMsg.m_sbyDirection = 0;
	m_sMsg.m_sbySensor    = 0;
	FPUT(DEV_101MD_BOX_ID,(BYTE*)&m_sMsg);
    #ifdef DEB_CKpModule
	Info("\n(__)CKPMM::>OUTT::%M",&m_sMsg);
    #endif
}
void CKpModule_Disconnect(This)
{
    DECLARE_MULTI_OPEN(CKpModule,CCyclicSystem)
	#ifdef DEB_CKpModule
	Info("\n(__)CKPMM::>Start DISCONNECT::>");
    #endif
	pT->m_blDiscStart = TRUE;
	pT->m_byDiscProc  = 0;
	//SendChar(PH_DISC0_REQ,"+");
	//SendChar(PH_DISC0_REQ,"+");
	//SendChar(PH_DISC0_REQ,"+");
	//pT->m_nDiscTMR.OnTimer(&pT->m_nDiscTMR,40);

	//SendCommand(PH_DISC0_REQ,"+++ ");
	//pT->m_nDiscTMR.OnTimer(&pT->m_nDiscTMR,20);
}
void CKpModule_StartCheck(This,BYTE byTime)
{
    DECLARE_MULTI_OPEN(CKpModule,CCyclicSystem)
	pT->m_nConnRepTMP.OnTimer(&pT->m_nConnRepTMP,byTime);
}
void CKpModule_StopCheck(This)
{
    DECLARE_MULTI_OPEN(CKpModule,CCyclicSystem)
	pT->m_nConnRepTMP.OfTimer(&pT->m_nConnRepTMP);
}
void CKpModule_SendObserveMsg(This)
{
    DECLARE_MULTI_OPEN(CKpModule,CCyclicSystem)
	CTeleSensor *pSN;
	if(pT->m_byObsObject<pT->m_wAmChannel)
	{
     pSN = pT->m_pTeleSensor[pT->m_byObsObject];
     pSN->SendObsrveMsg(pSN->pChld);
	 pT->m_nConnRepTMP.OnTimer(&pT->m_nConnRepTMP,pT->m_byObsTime);
	}
}
void CKpModule_SaveInPin(This)
{
    DECLARE_MULTI_OPEN(CKpModule,CCyclicSystem)
	CTeleSensor *pSN;WORD i;
	FFREE(BOX_L4_1);
	for (i=0;i<pT->m_wAmChannel;i++)
	{
		pSN = pT->m_pTeleSensor[i];
		pSN->SetInPinEvent(pSN->pChld);
	}
}
void CKpModule_SaveAlarmPin(This)
{
    DECLARE_MULTI_OPEN(CKpModule,CCyclicSystem)
	CTeleSensor *pSN;WORD i;
	FFREE(BOX_L4_1);
	for (i=0;i<pT->m_wAmChannel;i++)
	{
		pSN = pT->m_pTeleSensor[i];
		pSN->SaveAlarmPin(pSN->pChld);
	}
}

_GLOBAL INT nKPC,nKPC1;
void CKpModule_CyclicProc(This)
{
    DECLARE_MULTI_OPEN(CKpModule,CCyclicSystem)
	CTeleSensor *pSN;WORD i;

	if(pT->m_blDiscStart)
	{
	 if(++nKPC%10==0)
	 {
	  SendChar(PH_DISC0_REQ,"+");
	  if(++pT->m_byDiscProc==3)
	  {
	   pT->m_blDiscStart = FALSE;
	   pT->m_byDiscProc  = 0;
	   pT->m_nDiscTMR.OnTimer(&pT->m_nDiscTMR,20);
	  }
	 }
	}

	for (i=0;i<pT->m_wAmChannel;i++)
	{
     pSN = pT->m_pTeleSensor[i];
	 pSN->ObserveProc(pSN);
	}
    if (++nKPC1%20==0)pT->CheckSlot(pT);
	//if (++nKP%10==0)pT->CheckEventProc(pT);
	//Info("\n(%b)CKPMD::> CyclicProc",&pT->m_byKpID);
}
void CKpModule_CheckSlot(This)
{
    DECLARE_MULTI_OPEN(CKpModule,CCyclicSystem)
    BYTE i;
	BOOL *blpSlotState,blState=TRUE;
	for(i=0;i<pT->m_pComputer->m_bySlotAmout;i++)
	{
	 blpSlotState = (BOOL*)pT->m_pComputer->m_pvSlot[i]->m_pvAlmState;
	 if(*blpSlotState==FALSE) pT->m_pPCT->sSlot[i].byAlmState = 1;
	 if(*blpSlotState==TRUE)  pT->m_pPCT->sSlot[i].byAlmState = 0;
	}
}
BOOL CKpModule_SaveSlotState(This)
{
    DECLARE_MULTI_OPEN(CKpModule,CCyclicSystem)
	SKPEVENT sEV;
	//STSPARAM *pTS;
	//SHARDCOMPUTERTABLE *pH = pT->m_pPCT;
    BYTE i;
	for(i=0;i<pT->m_pComputer->m_bySlotAmout;i++)
	{
	 sEV.wLen    = sizeof(SKPEVENT);
	 sEV.byType  = REG_HARDT_ADDR;
     sEV.byCause = EV_ALS_CH;
	 sEV.byAddr  = i;
	 sEV.wValue  = (WORD)pT->m_pPCT->sSlot[i].byAlmState;
	 GetCurTime(&sEV.sTime);
	 FPUT1(BOX_L4_1,(BYTE*)&sEV);
	 #ifdef DEB_CTeleSensor
	 Info("\n(%b)CTLIN::>TP[%b]:AD[%b]:VL[%w]:CS[%s]:",&i,&sEV.byType,&sEV.byAddr,&sEV.wValue,STTS[sEV.byCause]);
     #endif
	}
	return TRUE;
}
BOOL CKpModule_Serialize(This,BOOL blDir)
{
	DECLARE_MULTI_OPEN(CKpModule,CCyclicSystem)
	BOOL res = TRUE;
	if (blDir==TRUE) res = pT->SaveContenst(pT);
	if (blDir==FALSE)res = pT->LoadContenst(pT);
	return res;
}
BOOL CKpModule_SaveContenst(This)
{
    DECLARE_MULTI_OPEN(CKpModule,CCyclicSystem)
	BOOL res = TRUE;
	pT->SaveTable(pT,&pT->m_nCT);
	//nValue_0++;
	if (!pT->m_pFlash->CompareMemory(pT->m_pFlash,(BYTE*)&pT->m_nCT,sizeof(SCONTENSTTABLE)))
	{
	 //nValue_1++;
	 if (!pT->m_pFlash->WriteFlash(pT->m_pFlash,(BYTE*)&pT->m_nCT,sizeof(SCONTENSTTABLE)))
 	 {
	 	//nValue_2++;
		res = FALSE;
	 }
	}
	return res;
}
_GLOBAL INT nWR0,nWR1,nWR2,nWR3;
BOOL CKpModule_LoadContenst(This)
{
    DECLARE_MULTI_OPEN(CKpModule,CCyclicSystem)
	BOOL res = FALSE;
	pT->m_nST.byKpID = 0xff;
	if (pT->m_pFlash->ReadFlash(pT->m_pFlash,(BYTE*)&pT->m_nST,sizeof(SCONTENSTTABLE)))
	{
		nWR0++;
	 if(pT->m_nST.byDefSett==1)
	 {
	 	nWR1++;
	 	 return FALSE;
	 }
	 if(pT->m_nST.byDefSett==0)
	 {
	  nWR2++;
	  if (pT->m_nST.byKpID==pT->m_byKpID)
	  {
	  nWR3++;
      pT->LoadTable(pT,&pT->m_nST);
	  res = TRUE;
	  }
	 }
	}
	return res;
}
void CKpModule_SaveTable(This,SCONTENSTTABLE *psTable)
{
    DECLARE_MULTI_OPEN(CKpModule,CCyclicSystem)
	psTable->byKpID = pT->m_byKpID;
    memcpy(&psTable->sKP ,&nKP ,sizeof(SKPPARAM));
	memcpy(&psTable->sARM,&nARM0,sizeof(SARMINTERFACE));
    memcpy(&psTable->sTI ,&nTI ,sizeof(STIPARAMS));
	memcpy(&psTable->sTS ,&nTS ,sizeof(STSPARAMS));
	memcpy(&psTable->sTU ,&nTU ,sizeof(STUPARAMS));
}
void CKpModule_LoadTable(This,SCONTENSTTABLE *psTable)
{
    DECLARE_MULTI_OPEN(CKpModule,CCyclicSystem)
	pT->m_byKpID = psTable->byKpID;
    memcpy(&nKP ,&psTable->sKP ,sizeof(SKPPARAM));
	memcpy(&nARM0,&psTable->sARM,sizeof(SARMINTERFACE));
    memcpy(&nTI ,&psTable->sTI ,sizeof(STIPARAMS));
	memcpy(&nTS ,&psTable->sTS ,sizeof(STSPARAMS));
	memcpy(&nTU ,&psTable->sTU ,sizeof(STUPARAMS));
}
void CKpModule_CKpModule(This)
{
    DECLARE_MULTI_OPEN(CKpModule,CCyclicSystem)
	DECLARE_REGISTRATION(CKpModule,Init)
	DECLARE_REGISTRATION(CKpModule,CreateChannels)
	DECLARE_REGISTRATION(CKpModule,StartConnect)
	DECLARE_REGISTRATION(CKpModule,Connect)
	DECLARE_REGISTRATION(CKpModule,Disconnect)
	DECLARE_REGISTRATION(CKpModule,DisconnectL2)
	DECLARE_REGISTRATION(CKpModule,CheckSlot)
	DECLARE_REGISTRATION(CKpModule,Serialize)
	DECLARE_REGISTRATION(CKpModule,SaveContenst)
	DECLARE_REGISTRATION(CKpModule,LoadContenst)
	DECLARE_REGISTRATION(CKpModule,SaveTable)
	DECLARE_REGISTRATION(CKpModule,LoadTable)
	DECLARE_REGISTRATION(CKpModule,SaveInPin)
	DECLARE_REGISTRATION(CKpModule,SaveAlarmPin)
	DECLARE_REGISTRATION(CKpModule,SaveSlotState)
	DECLARE_REGISTRATION(CKpModule,StartCheck)
	DECLARE_REGISTRATION(CKpModule,StopCheck)
	DECLARE_REGISTRATION(CKpModule,SendObserveMsg)
	DECLARE_VIRTUAL_FUNC(CKpModule,EventHandler)
	DECLARE_VIRTUAL_FUNC(CKpModule,CyclicProc)
}
void CKpModule_DCKpModule(This)
{
	DECLARE_MULTI_OPEN(CKpModule,CCyclicSystem)
}
DECLARE_MULTI_CREATE(CKpModule,CCyclicSystem)
```

#### bnraninput.c
```c
/********************************************************************
 * COPYRIGHT -- Kontora
 ********************************************************************
 * Program: bnrmain
 * File: bnrlsens.c
 * Author: Abramenya
 * Created: January 19, 2009
 *******************************************************************/

#include "bnraninput.h"
#ifdef _DEFAULT_INCLUDES
 #include <AsDefault.h>
#endif
//Analog Slot
#ifdef DEB_CAnIOSlot
SINT *chSlotType[] =
{
	"DEV_DEFAULT_PORT",
    "DEV_PLC_CPU_260",
	"DEV_PLC_CPU_X20",
	"DEV_TCPCOM_IF_681",
	"DEV_PWCOM_PS9500",
	"DEV_COM_CS1020",
	"DEV_AI_3AI375_6",
	"DEV_AI_X20AI4622",
	"DEV_AI_X20AI2622",
	"DEV_AO_3AO775_6",
	"DEV_AO_X20AO4622",
	"DEV_DI_3DI477_6",
	"DEV_DI_X20DM9371",
	"DEV_DI_X20DI9371",
	"DEV_DI_X20DI2377",
	"DEV_DO_3DO760_6",
	"DEV_DO_X20DM9322",
	"DEV_DO_X20DO9321",
	"DEV_AT_X20AT2222"
};
#endif
_GLOBAL INT iCAnIOSlotVal;
void CAnIOSlot_InitSlot(This,SHARDSLOT *pSlot)
{
	 CAnalogPin *pvPin;
	 BYTE i;
	 SHARDPIN sPin,sAlPin;
	 UINT **pInput;
	 BOOL **pAlInput;
	 DECLARE_MULTI_OPEN(CAnIOSlot,CSlot)
     #ifdef DEB_CAnIOSlot
	 Info("\n(%b)CANIN::>Create Slot:[%s]x%b.",&pSlot->bySlotNumber,chSlotType[pSlot->bySlotType],&pSlot->byPinAmout);
     #endif
	 iCAnIOSlotVal++;
	 pInput   = (UINT**)pSlot->pvPin;
	 pAlInput = (BOOL**)pSlot->pvAlmPin;

	 if(pSlot->byPinAmout>0)
	 {
	  for(i=0;i<pSlot->byPinAmout;i++)
	  {
		pvPin = &pT->m_pPin[i];
		sPin.byPinNumber = i;
		sPin.byPinState  = PIN_STATE_OFF;
		sPin.pvValue     = (PVOID)pInput[i];

		sAlPin.byPinNumber = i;
		sAlPin.byPinState  = PIN_STATE_OFF;
		sAlPin.pvValue     = (PVOID)pAlInput[i];

		if(pvPin!=NULL)
		{
 		 InitObject(CAnalogPin,pvPin);
		 pvPin->pBase->SetSlot(pvPin->pBase,pB->m_bySlotNumber);
		 pvPin->pBase->Init(pvPin->pBase,&sPin,&sAlPin);
		}
	  }
	 }
}
void CAnIOSlot_Connect(This,CAnalogPin *pPin)
{
     DECLARE_MULTI_OPEN(CAnIOSlot,CSlot)
}
CPin* CAnIOSlot_GetPin(This,BYTE byNumber)
{
     DECLARE_MULTI_OPEN(CAnIOSlot,CSlot)
	 if(byNumber<pB->m_byAmPin)
     return pT->m_pPin[byNumber].pBase;
	 return NULL;
}
void CAnIOSlot_CAnIOSlot(This)
{
     DECLARE_MULTI_OPEN(CAnIOSlot,CSlot)
	 DECLARE_REGISTRATION(CAnIOSlot,Connect)
	 DECLARE_VIRTUAL_FUNC(CAnIOSlot,InitSlot)
	 DECLARE_VIRTUAL_FUNC(CAnIOSlot,GetPin)
}
void CAnIOSlot_DCAnIOSlot(This)
{
	 DECLARE_MULTI_OPEN(CAnIOSlot,CSlot)
}
DECLARE_MULTI_CREATE(CAnIOSlot,CSlot)
//Analog Slot 4
void CAnIOSlot4_InitSlot(This,SHARDSLOT *pSlot)
{
	 CAnalogPin *pvPin;
	 BYTE i;
	 SHARDPIN sPin,sAlPin;
	 UINT **pInput;
	 BOOL **pAlInput;
	 DECLARE_MULTI_OPEN(CAnIOSlot4,CSlot)
     #ifdef DEB_CAnIOSlot
	 Info("\n(%b)CANIN::>Create Slot:[%s]x%b.",&pSlot->bySlotNumber,chSlotType[pSlot->bySlotType],&pSlot->byPinAmout);
     #endif
	 iCAnIOSlotVal++;
	 pInput   = (UINT**)pSlot->pvPin;
	 pAlInput = (BOOL**)pSlot->pvAlmPin;
	 if(pSlot->byPinAmout>0)
	 {
	  for(i=0;i<pSlot->byPinAmout;i++)
	  {
		pvPin = &pT->m_pPin[i];
		sPin.byPinNumber = i;
		sPin.byPinState  = PIN_STATE_OFF;
		sPin.pvValue     = (PVOID)pInput[i];

		sAlPin.byPinNumber = i;
		sAlPin.byPinState  = PIN_STATE_OFF;
		sAlPin.pvValue     = (PVOID)pAlInput[i];

		if(pvPin!=NULL)
		{
 		 InitObject(CAnalogPin,pvPin);
		 pvPin->pBase->SetSlot(pvPin->pBase,pB->m_bySlotNumber);
		 pvPin->pBase->Init(pvPin->pBase,&sPin,&sAlPin);
		}
	  }
	 }
}
void CAnIOSlot4_Connect(This,CAnalogPin *pPin)
{
     DECLARE_MULTI_OPEN(CAnIOSlot4,CSlot)
}
CPin* CAnIOSlot4_GetPin(This,BYTE byNumber)
{
     DECLARE_MULTI_OPEN(CAnIOSlot4,CSlot)
	 if(byNumber<pB->m_byAmPin)
     return pT->m_pPin[byNumber].pBase;
	 return NULL;
}
void CAnIOSlot4_CAnIOSlot4(This)
{
     DECLARE_MULTI_OPEN(CAnIOSlot4,CSlot)
	 DECLARE_REGISTRATION(CAnIOSlot4,Connect)
	 DECLARE_VIRTUAL_FUNC(CAnIOSlot4,InitSlot)
	 DECLARE_VIRTUAL_FUNC(CAnIOSlot4,GetPin)
}
void CAnIOSlot4_DCAnIOSlot4(This)
{
	 DECLARE_MULTI_OPEN(CAnIOSlot4,CSlot)
}
DECLARE_MULTI_CREATE(CAnIOSlot4,CSlot)
//Digital Slot
void CDgIOSlot_InitSlot(This,SHARDSLOT *pSlot)
{
	 CDigitalPin *pvPin;
	 BYTE i;
	 BOOL **pInput,**pAlInput;
	 SHARDPIN sPin,sAlPin;
	 DECLARE_MULTI_OPEN(CDgIOSlot,CSlot)
	 #ifdef DEB_CDgIOSlot
     Info("\n(%b)CDGIN::>Create Slot:[%s]x%b.",&pSlot->bySlotNumber,chSlotType[pSlot->bySlotType],&pSlot->byPinAmout);
     #endif
	 pInput   = (BOOL**)pSlot->pvPin;
	 pAlInput = (BOOL**)pSlot->pvAlmPin;
	 if(pSlot->byPinAmout>0)
	 {
	  for(i=0;i<pSlot->byPinAmout;i++)
	  {
		  pvPin = &pT->m_pPin[i];
		  sPin.byPinNumber = i;
		  //sPin.byPinType   = PIN_DG_INOT_BOL;
		  sPin.byPinState  = PIN_STATE_OFF;
		  sPin.pvValue     = (PVOID)pInput[i];

		  sAlPin.byPinState  = PIN_STATE_OFF;
		  sAlPin.pvValue     = (PVOID)pAlInput[i];
		  sAlPin.byPinNumber = i;
		  if(pvPin!=NULL)
		  {
		   InitObject(CDigitalPin,pvPin);
		   pvPin->pBase->SetSlot(pvPin->pBase,pB->m_bySlotNumber);
		   pvPin->pBase->Init(pvPin->pBase,&sPin,&sAlPin);
		  }
	  }
	 }
}
void CDgIOSlot_Connect(This,CDigitalPin *pPin)
{
	 DECLARE_MULTI_OPEN(CDgIOSlot,CSlot)
	 //pT->m_pPin[pPin->pBase->m_byPinNumber] = pPin;
}
CPin* CDgIOSlot_GetPin(This,BYTE byNumber)
{
	 DECLARE_MULTI_OPEN(CDgIOSlot,CSlot)
	 if(byNumber<pB->m_byAmPin)
	 return pT->m_pPin[byNumber].pBase;
	 return NULL;
}
void CDgIOSlot_CDgIOSlot(This)
{
	 DECLARE_MULTI_OPEN(CDgIOSlot,CSlot)
	 DECLARE_REGISTRATION(CDgIOSlot,Connect)
  	 DECLARE_VIRTUAL_FUNC(CDgIOSlot,InitSlot)
	 DECLARE_VIRTUAL_FUNC(CDgIOSlot,GetPin)
}
void CDgIOSlot_DCDgIOSlot(This)
{
	 DECLARE_MULTI_OPEN(CDgIOSlot,CSlot)
}
DECLARE_MULTI_CREATE(CDgIOSlot,CSlot)
//CountSlot Slot
void CCountSlot_InitSlot(This,SHARDSLOT *pSlot)
{
	CDCounterPin *pvPin;
	BYTE i;
	BOOL **pInput,**pAlInput;
	SHARDPIN sPin,sAlPin;
	DECLARE_MULTI_OPEN(CCountSlot,CSlot)
    #ifdef DEB_CDgIOSlot
		Info("\n(%b)CDGIN::>Create Slot:[%s]x%b.",&pSlot->bySlotNumber,chSlotType[pSlot->bySlotType],&pSlot->byPinAmout);
    #endif
	pInput   = (BOOL**)pSlot->pvPin;
	pAlInput = (BOOL**)pSlot->pvAlmPin;
	if(pSlot->byPinAmout>0)
	{
		for(i=0;i<pSlot->byPinAmout;i++)
		{
			pvPin = &pT->m_pPin[i];
			sPin.byPinNumber = i;
			//sPin.byPinType   = PIN_DG_INOT_BOL;
			sPin.byPinState  = PIN_STATE_OFF;
			sPin.pvValue     = (PVOID)pInput[i];

			sAlPin.byPinState  = PIN_STATE_OFF;
			sAlPin.pvValue     = (PVOID)pAlInput[i];
			sAlPin.byPinNumber = i;
			if(pvPin!=NULL)
			{
				InitObject(CDCounterPin,pvPin);
				pvPin->pBase->SetSlot(pvPin->pBase,pB->m_bySlotNumber);
				pvPin->pBase->Init(pvPin->pBase,&sPin,&sAlPin);
			}
		}
	}
}
void CCountSlot_Connect(This,CDCounterPin *pPin)
{
	DECLARE_MULTI_OPEN(CCountSlot,CSlot)
	//pT->m_pPin[pPin->pBase->m_byPinNumber] = pPin;
}
CPin* CCountSlot_GetPin(This,BYTE byNumber)
{
	DECLARE_MULTI_OPEN(CCountSlot,CSlot)
	if(byNumber<pB->m_byAmPin)
	return pT->m_pPin[byNumber].pBase;
	return NULL;
}
void CCountSlot_CCountSlot(This)
{
	DECLARE_MULTI_OPEN(CCountSlot,CSlot)
	DECLARE_REGISTRATION(CCountSlot,Connect)
	DECLARE_VIRTUAL_FUNC(CCountSlot,InitSlot)
	DECLARE_VIRTUAL_FUNC(CCountSlot,GetPin)
}
void CCountSlot_DCCountSlot(This)
{
	DECLARE_MULTI_OPEN(CCountSlot,CSlot)
}
DECLARE_MULTI_CREATE(CCountSlot,CSlot)
//CountSlot Slot
void CTemperatureSlot_InitSlot(This,SHARDSLOT *pSlot)
{
	CTemperaturePin *pvPin;
	BYTE i;
	BOOL **pInput,**pAlInput;
	SHARDPIN sPin,sAlPin;
	DECLARE_MULTI_OPEN(CTemperatureSlot,CSlot)
    #ifdef DEB_CDgIOSlot
	Info("\n(%b)CDGIN::>Create Slot:[%s]x%b.",&pSlot->bySlotNumber,chSlotType[pSlot->bySlotType],&pSlot->byPinAmout);
    #endif
	pInput   = (BOOL**)pSlot->pvPin;
	pAlInput = (BOOL**)pSlot->pvAlmPin;
	if(pSlot->byPinAmout>0)
	{
		for(i=0;i<pSlot->byPinAmout;i++)
		{
			pvPin = &pT->m_pPin[i];
			sPin.byPinNumber = i;
			//sPin.byPinType   = PIN_DG_INOT_BOL;
			sPin.byPinState  = PIN_STATE_OFF;
			sPin.pvValue     = (PVOID)pInput[i];

			sAlPin.byPinState  = PIN_STATE_OFF;
			sAlPin.pvValue     = (PVOID)pAlInput[i];
			sAlPin.byPinNumber = i;
			if(pvPin!=NULL)
			{
				InitObject(CTemperaturePin,pvPin);
				pvPin->pBase->SetSlot(pvPin->pBase,pB->m_bySlotNumber);
				pvPin->pBase->Init(pvPin->pBase,&sPin,&sAlPin);
			}
		}
	}
}
void CTemperatureSlot_Connect(This,CDCounterPin *pPin)
{
	DECLARE_MULTI_OPEN(CTemperatureSlot,CSlot)
	//pT->m_pPin[pPin->pBase->m_byPinNumber] = pPin;
}
CPin* CTemperatureSlot_GetPin(This,BYTE byNumber)
{
	DECLARE_MULTI_OPEN(CTemperatureSlot,CSlot)
	if(byNumber<pB->m_byAmPin)
	return pT->m_pPin[byNumber].pBase;
	return NULL;
}
void CTemperatureSlot_CTemperatureSlot(This)
{
	DECLARE_MULTI_OPEN(CTemperatureSlot,CSlot)
	DECLARE_REGISTRATION(CTemperatureSlot,Connect)
	DECLARE_VIRTUAL_FUNC(CTemperatureSlot,InitSlot)
	DECLARE_VIRTUAL_FUNC(CTemperatureSlot,GetPin)
}
void CTemperatureSlot_DCTemperatureSlot(This)
{
	DECLARE_MULTI_OPEN(CTemperatureSlot,CSlot)
}
DECLARE_MULTI_CREATE(CTemperatureSlot,CSlot)
```

#### bnrauto.c
```c
/********************************************************************
 * COPYRIGHT -- Kontora
 ********************************************************************
 * Program: bnrmain
 * File: bnrlsens.c
 * Author: Abramenya
 * Created: January 19, 2009
 *******************************************************************/
#include "bnrauto.h"
#ifdef _DEFAULT_INCLUDES
 #include <AsDefault.h>
#endif
DECLARE_TASKCHAIN(Skip)
{
    {EXIT_D}
};
DECLARE_STATE(BadState)
{
    {EV_UNKNOWN_REQ, Skip}
};
DECLARE_STATELIST(StateList)
{
    {S_BAD, BadState}
};
BOOL CAuto_SetState(This,TStateCode vNewState)
{
	DECLARE_SINGLE_OPEN(CAuto)
    TStateList * pvList = pT->GetStateList(pC);
    pT->m_pvState = pvList[(INT16)vNewState].m_pvState;
    pT->m_vState  = vNewState;
	pT->v[STATE] = vNewState;
    return TRUE;
}
BOOL CAuto_HandleEvent(This,TEvent vEvent)
{
	DECLARE_SINGLE_OPEN(CAuto)
	TState* pvState;
    for(pvState=pT->m_pvState; pvState->m_vEvent!=EV_UNKNOWN_REQ; pvState++)
    {
        if(pvState->m_vEvent==vEvent)
        {
            return pT->HandleTask(pC,pvState->m_pvTask);
        }
    }
    return FALSE;
}
BOOL CAuto_HandleTask(This,TTask* pvTask)
{
	DECLARE_SINGLE_OPEN(CAuto)
    return (*pvTask==EXIT_D)?TRUE:FALSE;
}
TStateList* CAuto_GetStateList(This)
{
	DECLARE_SINGLE_OPEN(CAuto)
    return (TStateList*)&StateList;
}
TStateCode CAuto_GetStateCode(This)
{
	DECLARE_SINGLE_OPEN(CAuto)
	return pT->m_vState;
}
TState* CAuto_GetState(This)
{
	DECLARE_SINGLE_OPEN(CAuto)
	return pT->m_pvState;
}
void CAuto_CAuto(This)
{
    DECLARE_SINGLE_OPEN(CAuto)
	DECLARE_REGISTRATION(CAuto,GetStateList)
	DECLARE_REGISTRATION(CAuto,HandleTask)
	DECLARE_REGISTRATION(CAuto,HandleEvent)
	DECLARE_REGISTRATION(CAuto,SetState)
	DECLARE_REGISTRATION(CAuto,GetStateCode)
	DECLARE_REGISTRATION(CAuto,GetState)
    pT->m_pvState = BadState;
    pT->m_vState  = S_BAD;
}
void CAuto_DCAuto(This)
{
	DECLARE_SINGLE_OPEN(CAuto)
}
DECLARE_SINGLE_CREATE(CAuto)
```

#### bnrchains.c
```c
/********************************************************************
 * COPYRIGHT -- Kontora
 ********************************************************************
 * Program: bnrmain
 * File: bnrchains.h
 * Author: Abramenya
 * Created: February 04, 2009
 *******************************************************************/
#ifndef WIN32
#include <bur/plctypes.h>
#endif
#include "typedefs.h"
#include "bnrconst.h"
//Обработчик событий датчика уровня(два выхода) для АС1-3
IMPORT_TASKCHAIN(Skip);
//пустое состояние
IMPORT_STATE(BadState);
/*
IMPORT_STATELIST(STL_LV00_SENS);//2-Out
IMPORT_STATELIST(STL_PS00_SENS);//2-Out
IMPORT_STATELIST(STL_TM00_SENS);//1-Out
IMPORT_STATELIST(STL_LV04_SENS);//1-Out
IMPORT_STATELIST(STL_LVN4_SENS);//0-Out
IMPORT_STATELIST(STL_PS04_SENS);//1-Out
*/
//Gate Logic///////////////////////////////////////
DECLARE_TASKCHAIN(Lv00LoOperGate)
{
	//CMD_OPENGATE,GT0,80,
	//CMD_OPENGATE,GT1,20,
	//CMD_SETVALUE,INC_INP,1,
	CMD_SETSTATE,SNS_STATE_FREE,
	EXIT_D,
};
DECLARE_TASKCHAIN(Lv00HiOperGate)
{
	//CMD_OPENGATE,GT0,20,
	//CMD_OPENGATE,GT1,80,
	//CMD_SETVALUE,INC_INP,0,
	CMD_SETSTATE,SNS_STATE_FREE,
	EXIT_D,
};
//Alarm Logic///////////////////////////////////////
DECLARE_TASKCHAIN(Lv00SetAlmHilev)
{
	//CMD_TIMERON ,TMR_SET_ALM_HI,T5SEC,
	//CMD_TIMEROFF,TMR_REM_ALM_HI,
	//CMD_SETSTATE,SNS_STATE_FREE,
	EXIT_D,
};
DECLARE_TASKCHAIN(Lv00RemAlmHiLev)
{
	//CMD_TIMERON ,TMR_REM_ALM_HI,T5SEC,
	//CMD_TIMEROFF,TMR_SET_ALM_HI,
	//CMD_SETSTATE,SNS_STATE_FREE,
	EXIT_D,
};
DECLARE_TASKCHAIN(Lv00SetAlmLolev)
{
	//CMD_TIMERON ,TMR_SET_ALM_LO,T5SEC,
	//CMD_TIMEROFF,TMR_REM_ALM_LO,
	//CMD_SETSTATE,SNS_STATE_FREE,
	EXIT_D,
};
DECLARE_TASKCHAIN(Lv00RemAlmLolev)
{
	//CMD_TIMERON ,TMR_REM_ALM_LO,T5SEC,
	//CMD_TIMEROFF,TMR_SET_ALM_LO,
	//CMD_SETSTATE,SNS_STATE_FREE,
	EXIT_D,
};
/////////////////////////////////////////
DECLARE_TASKCHAIN(Lv00TmrSetAlmHilev)
{
	CMD_SEND,MDL_ADMIN,EV_ADMIN_SET_ALM_HILEV_REQ,
	//CMD_SETSTATE,SNS_STATE_FREE,
	EXIT_D,
};
DECLARE_TASKCHAIN(Lv00TmrRemAlmHiLev)
{
	CMD_SEND,MDL_ADMIN,EV_ADMIN_REM_ALM_HILEV_REQ,
	//CMD_SETSTATE,SNS_STATE_FREE,
	EXIT_D,
};
DECLARE_TASKCHAIN(Lv00TmrSetAlmLolev)
{
    CMD_SEND,MDL_ADMIN,EV_ADMIN_SET_ALM_LOLEV_REQ,
	//CMD_SETSTATE,SNS_STATE_FREE,
	EXIT_D,
};
DECLARE_TASKCHAIN(Lv00TmrRemAlmLolev)
{
	CMD_SEND,MDL_ADMIN,EV_ADMIN_REM_ALM_LOLEV_REQ,
	//CMD_SETSTATE,SNS_STATE_FREE,
	EXIT_D,
};
/////////////////////////////////////////
DECLARE_STATE(Lv00StateFree)
{
    { EV_ADMIN_OPER_LO_REQ,            Lv00LoOperGate     },
    { EV_ADMIN_OPER_HI_REQ,            Lv00HiOperGate     },
    { EV_ADMIN_SET_ALM_HILEV_REQ,      Lv00SetAlmHilev    },
    { EV_ADMIN_REM_ALM_HILEV_REQ,      Lv00RemAlmHiLev    },
    { EV_ADMIN_SET_ALM_LOLEV_REQ,      Lv00SetAlmLolev    },
    { EV_ADMIN_REM_ALM_LOLEV_REQ,      Lv00RemAlmLolev    },
    { EV_SENSR_TMR_SAHI,               Lv00TmrSetAlmHilev },
    { EV_SENSR_TMR_RAHI,               Lv00TmrRemAlmHiLev },
    { EV_SENSR_TMR_SALO,               Lv00TmrSetAlmLolev },
    { EV_SENSR_TMR_RALO,               Lv00TmrRemAlmLolev },
    { EV_UNKNOWN_REQ,                  Skip               }
};
DECLARE_STATELIST(STL_LV00_SENS)
{
    { SNS_STATE_FREE,            Lv00StateFree   },
    { S_BAD,                     BadState        }
};
//Обработчик событий датчика давления(два выхода) для АС1-3
//Gate Logic///////////////////////////////////////
DECLARE_TASKCHAIN(Ps00LoOperGate)
{
	CMD_SETSTATE,SNS_STATE_FREE,
	EXIT_D,
};
DECLARE_TASKCHAIN(Ps00HiOperGate)
{
	CMD_SETSTATE,SNS_STATE_FREE,
	EXIT_D,
};
DECLARE_STATE(Ps00StateFree)
{
    { EV_ADMIN_OPER_LO_REQ,            Ps00LoOperGate     },
    { EV_ADMIN_OPER_HI_REQ,            Ps00HiOperGate     },
    { EV_ADMIN_SET_ALM_HILEV_REQ,      Lv00SetAlmHilev    },
    { EV_ADMIN_REM_ALM_HILEV_REQ,      Lv00RemAlmHiLev    },
    { EV_ADMIN_SET_ALM_LOLEV_REQ,      Lv00SetAlmLolev    },
    { EV_ADMIN_REM_ALM_LOLEV_REQ,      Lv00RemAlmLolev    },
    { EV_SENSR_TMR_SAHI,               Lv00TmrSetAlmHilev },
    { EV_SENSR_TMR_RAHI,               Lv00TmrRemAlmHiLev },
    { EV_SENSR_TMR_SALO,               Lv00TmrSetAlmLolev },
    { EV_SENSR_TMR_RALO,               Lv00TmrRemAlmLolev },
    { EV_UNKNOWN_REQ,                  Skip               }
};
DECLARE_STATELIST(STL_PS00_SENS)
{
    { SNS_STATE_FREE,                  Ps00StateFree      },
    { S_BAD,                           BadState           }
};
//Обработчик событий датчика температуры(один выход) для АС1-4
//Gate Logic///////////////////////////////////////
DECLARE_TASKCHAIN(Tm00LoOperGate)
{
	CMD_SETSTATE,SNS_STATE_FREE,
	EXIT_D,
};
DECLARE_TASKCHAIN(Tm00HiOperGate)
{
	CMD_SETSTATE,SNS_STATE_FREE,
	EXIT_D,
};
DECLARE_STATE(Tm00StateFree)
{
    { EV_ADMIN_OPER_LO_REQ,            Tm00LoOperGate     },
    { EV_ADMIN_OPER_HI_REQ,            Tm00HiOperGate     },
    { EV_ADMIN_SET_ALM_HILEV_REQ,      Lv00SetAlmHilev    },
    { EV_ADMIN_REM_ALM_HILEV_REQ,      Lv00RemAlmHiLev    },
    { EV_ADMIN_SET_ALM_LOLEV_REQ,      Lv00SetAlmLolev    },
    { EV_ADMIN_REM_ALM_LOLEV_REQ,      Lv00RemAlmLolev    },
    { EV_SENSR_TMR_SAHI,               Lv00TmrSetAlmHilev },
    { EV_SENSR_TMR_RAHI,               Lv00TmrRemAlmHiLev },
    { EV_SENSR_TMR_SALO,               Lv00TmrSetAlmLolev },
    { EV_SENSR_TMR_RALO,               Lv00TmrRemAlmLolev },
    { EV_UNKNOWN_REQ,                  Skip               }
};
DECLARE_STATELIST(STL_TM00_SENS)
{
    { SNS_STATE_FREE,                  Tm00StateFree      },
    { S_BAD,                           BadState           }
};
//Обработчик событий датчика уровня(два выхода) для АС4
//Gate Logic///////////////////////////////////////
DECLARE_TASKCHAIN(Lv04LoOperGate)
{
	CMD_OPENGATE,GT0,90,
	CMD_OPENGATE,GT1,30,
	CMD_SETVALUE,INC_INP,1,
	CMD_SETSTATE,SNS_STATE_FREE,
	EXIT_D,
};
DECLARE_TASKCHAIN(Lv04HiOperGate)
{
	CMD_OPENGATE,GT0,30,
	CMD_OPENGATE,GT1,90,
	CMD_SETVALUE,INC_INP,0,
	CMD_SETSTATE,SNS_STATE_FREE,
	EXIT_D,
};
DECLARE_STATE(Lv04StateFree)
{
    { EV_ADMIN_OPER_LO_REQ,            Lv04LoOperGate     },
    { EV_ADMIN_OPER_HI_REQ,            Lv04HiOperGate     },
    { EV_ADMIN_SET_ALM_HILEV_REQ,      Lv00SetAlmHilev    },
    { EV_ADMIN_REM_ALM_HILEV_REQ,      Lv00RemAlmHiLev    },
    { EV_ADMIN_SET_ALM_LOLEV_REQ,      Lv00SetAlmLolev    },
    { EV_ADMIN_REM_ALM_LOLEV_REQ,      Lv00RemAlmLolev    },
    { EV_SENSR_TMR_SAHI,               Lv00TmrSetAlmHilev },
    { EV_SENSR_TMR_RAHI,               Lv00TmrRemAlmHiLev },
    { EV_SENSR_TMR_SALO,               Lv00TmrSetAlmLolev },
    { EV_SENSR_TMR_RALO,               Lv00TmrRemAlmLolev },
    { EV_UNKNOWN_REQ,                  Skip               }
};
DECLARE_STATELIST(STL_LV04_SENS)
{
    { SNS_STATE_FREE,                  Lv04StateFree      },
    { S_BAD,                           BadState           }
};
//Обработчик событий датчика уровня(нет выхода) для АС4
DECLARE_STATELIST(STL_LVN4_SENS)
{
    { SNS_STATE_FREE,                  Tm00StateFree      }, //Как для температуры
    { S_BAD,                           BadState           }
};
//Обработчик событий датчика давления(один выход) для АС4
DECLARE_STATELIST(STL_PS04_SENS)
{
    { SNS_STATE_FREE,                  Tm00StateFree      }, //Как для температуры
    { S_BAD,                           BadState           }
};
```

#### bnrcomputer.c
```c
/********************************************************************
 * COPYRIGHT -- Kontora
 ********************************************************************
 * Program: bnrmain
 * File: bnrlsens.c
 * Author: Abramenya
 * Created: January 19, 2009
 *******************************************************************/

#include "bnrcomputer.h"
#ifdef _DEFAULT_INCLUDES
 #include <AsDefault.h>
#endif
void CComputer_Init(This,SHARDCOMPUTERTABLE *pTable)
{
    DECLARE_SINGLE_OPEN(CComputer)
    #ifdef DEB_CComputer
	Info("\n(__)CCOMP::>Create Computer:%s:%s",pTable->chComputerName,pTable->chDateOfWrite);
    #endif
	pT->InitDevModule(pT,pTable);
}
void CComputer_InitDevModule(This,SHARDCOMPUTERTABLE *pTable)
{
	int i;
	CSlot *m_pSlot;
    DECLARE_SINGLE_OPEN(CComputer)
	New(sizeof(SHARDCOMPUTERTABLE),pT->m_pConfigTable);
	memcpy(pT->m_pConfigTable,pTable,sizeof(SHARDCOMPUTERTABLE));
	pT->m_byComputerType = pTable->byComputerType;
	pT->m_bySlotAmout = pTable->bySlotAmout;
	strcpy(pT->m_chProgrammVersion,pTable->chProgrammVersion);
	strcpy(pT->m_chComputerName,pTable->chComputerName);
	strcpy(pT->m_chDateOfWrite,pTable->chDateOfWrite);
	New(sizeof(CSlot*)*pTable->bySlotAmout,pT->m_pvSlot);
	for(i=0;i<pTable->bySlotAmout;i++)
	{
		m_pSlot = pT->CreateSlot(pT,&pTable->sSlot[i]);
		if(m_pSlot!=NULL)
			pT->Connect(pT,m_pSlot);
	}
}
CSlot* CComputer_CreateSlot(This,SHARDSLOT *psvSlot)
{
    DECLARE_SINGLE_OPEN(CComputer)
	switch(psvSlot->bySlotType)
	{
	   case DEV_PLC_CPU_260:
	   case DEV_PLC_CPU_X20:
            return pT->CreateSlotCPU_260(pT,psvSlot);
       case DEV_TCPCOM_IF_681:
            return pT->CreateSlotIF_681(pT,psvSlot);
	   case DEV_AI_3AI375_6:
		    return pT->CreateSlot3AI375_6(pT,psvSlot);
	   case DEV_DI_X20DI2377:
		    return pT->CreateSlotDI2377(pT,psvSlot);
       case DEV_AI_X20AI2622:
		    return pT->CreateSlot3AI375_6(pT,psvSlot);
	   case DEV_AT_X20AT2222:
		    return pT->CreateSlotAT2222(pT,psvSlot);
	   case DEV_AI_X20AI4622:
	   case DEV_AO_X20AO4622:
		    return pT->CreateSlot3AI4622(pT,psvSlot);
	   case DEV_AO_3AO775_6:
	    	return pT->CreateSlot3AO775_6(pT,psvSlot);
	   case DEV_DI_3DI477_6:
	   case DEV_DI_X20DI9371:
	   case DEV_DI_X20DM9371:
		    return pT->CreateSlot3DI477_6(pT,psvSlot);
	   case DEV_DO_3DO760_6:
	   case DEV_DO_X20DM9322:
	   case DEV_DO_X20DO9321:
		    return pT->CreateSlot3DO477_6(pT,psvSlot);
	   default:
	   break;
	}
    return NULL;
}
CSlot* CComputer_CreateSlotCPU_260(This,SHARDSLOT *psvSlot)
{
	 CDgIOSlot *pHSlot;
     DECLARE_SINGLE_OPEN(CComputer)
	 New(sizeof(CDgIOSlot),pHSlot);
	 InitObject(CDgIOSlot,pHSlot);
	 if (pHSlot!=NULL)
	 {
		pHSlot->pBase->Init(pHSlot->pBase,psvSlot);
	 }else return NULL;
	 return pHSlot->pBase;
}
CSlot* CComputer_CreateSlotIF_681(This,SHARDSLOT *psvSlot)
{
	 CDgIOSlot *pHSlot;
	 DECLARE_SINGLE_OPEN(CComputer)
	 New(sizeof(CDgIOSlot),pHSlot);
	 InitObject(CDgIOSlot,pHSlot);
	 if (pHSlot!=NULL)
	 {
		pHSlot->pBase->Init(pHSlot->pBase,psvSlot);
	 }else return NULL;
	 return pHSlot->pBase;
}
CSlot* CComputer_CreateSlot3DI477_6(This,SHARDSLOT *psvSlot)
{
	 CDgIOSlot *pHSlot;
	 DECLARE_SINGLE_OPEN(CComputer)
	 New(sizeof(CDgIOSlot),pHSlot);
	 InitObject(CDgIOSlot,pHSlot);
	 if (pHSlot!=NULL)
	 {
		pHSlot->pBase->Init(pHSlot->pBase,psvSlot);
	 }else return NULL;
	 return pHSlot->pBase;
}
CSlot* CComputer_CreateSlot3DO477_6(This,SHARDSLOT *psvSlot)
{
	 CDgIOSlot *pHSlot;
	 DECLARE_SINGLE_OPEN(CComputer)
	 New(sizeof(CDgIOSlot),pHSlot);
	 InitObject(CDgIOSlot,pHSlot);
	 if (pHSlot!=NULL)
	 {
		pHSlot->pBase->Init(pHSlot->pBase,psvSlot);
	 }else return NULL;
	 return pHSlot->pBase;
}
CSlot* CComputer_CreateSlot3AI375_6(This,SHARDSLOT *psvSlot)
{
	 CAnIOSlot *pHSlot;
	 DECLARE_SINGLE_OPEN(CComputer)
	 New(sizeof(CAnIOSlot),pHSlot);
	 InitObject(CAnIOSlot,pHSlot);
	 if (pHSlot!=NULL)
	 {
		pHSlot->pBase->Init(pHSlot->pBase,psvSlot);
	 }else return NULL;
	 return pHSlot->pBase;
}
CSlot* CComputer_CreateSlotAT2222(This,SHARDSLOT *psvSlot)
{
	CTemperatureSlot *pHSlot;
	DECLARE_SINGLE_OPEN(CComputer)
	New(sizeof(CTemperatureSlot),pHSlot);
	InitObject(CTemperatureSlot,pHSlot);
	if (pHSlot!=NULL)
	{
	   pHSlot->pBase->Init(pHSlot->pBase,psvSlot);
	}else return NULL;
	return pHSlot->pBase;
}
CSlot* CComputer_CreateSlotDI2377(This,SHARDSLOT *psvSlot)
{
	CCountSlot *pHSlot;
	DECLARE_SINGLE_OPEN(CComputer)
	New(sizeof(CCountSlot),pHSlot);
	InitObject(CCountSlot,pHSlot);
	if (pHSlot!=NULL)
	{
		pHSlot->pBase->Init(pHSlot->pBase,psvSlot);
	}else return NULL;
	return pHSlot->pBase;
}
CSlot* CComputer_CreateSlot3AI4622(This,SHARDSLOT *psvSlot)
{
	 CAnIOSlot4 *pHSlot;
	 DECLARE_SINGLE_OPEN(CComputer)
	 New(sizeof(CAnIOSlot4),pHSlot);
	 InitObject(CAnIOSlot4,pHSlot);
	 if (pHSlot!=NULL)
	 {
		pHSlot->pBase->Init(pHSlot->pBase,psvSlot);
	 }else return NULL;
	 return pHSlot->pBase;
}
CSlot* CComputer_CreateSlot3AO775_6(This,SHARDSLOT *psvSlot)
{
	 CAnIOSlot *pHSlot;
	 DECLARE_SINGLE_OPEN(CComputer)
	 New(sizeof(CAnIOSlot),pHSlot);
	 InitObject(CAnIOSlot,pHSlot);
	 if (pHSlot!=NULL)
	 {
		pHSlot->pBase->Init(pHSlot->pBase,psvSlot);
	 }else return NULL;
	 return pHSlot->pBase;
}
void CComputer_Connect(This,CSlot *pSlot)
{
     DECLARE_SINGLE_OPEN(CComputer);
     pT->m_pvSlot[pSlot->m_bySlotNumber] = pSlot->pThis;
}
CSlot* CComputer_GetSlot(This,BYTE byNumber)
{
     DECLARE_SINGLE_OPEN(CComputer)
	 if(byNumber < pT->m_pConfigTable->bySlotAmout)
     return pT->m_pvSlot[byNumber];
	 return NULL;
}
void CComputer_CComputer(This)
{
     DECLARE_SINGLE_OPEN(CComputer)
	 DECLARE_REGISTRATION(CComputer,Init)
	 DECLARE_REGISTRATION(CComputer,InitDevModule)
	 DECLARE_REGISTRATION(CComputer,Connect)
	 DECLARE_REGISTRATION(CComputer,CreateSlot)
	 DECLARE_REGISTRATION(CComputer,CreateSlotCPU_260)
	 DECLARE_REGISTRATION(CComputer,CreateSlotIF_681)
	 DECLARE_REGISTRATION(CComputer,CreateSlot3DI477_6)
	 DECLARE_REGISTRATION(CComputer,CreateSlot3DO477_6)
	 DECLARE_REGISTRATION(CComputer,CreateSlot3AI375_6)
	 DECLARE_REGISTRATION(CComputer,CreateSlot3AI4622)
	 DECLARE_REGISTRATION(CComputer,CreateSlotAT2222)
	 DECLARE_REGISTRATION(CComputer,CreateSlotDI2377)
	 DECLARE_REGISTRATION(CComputer,CreateSlot3AO775_6)
	 DECLARE_REGISTRATION(CComputer,GetSlot)
}
void CComputer_DCComputer(This)
{
	DECLARE_SINGLE_OPEN(CComputer)
	BYTE i;
	for(i=0;i<pT->m_bySlotAmout;i++)
	{
	 switch(pT->m_pvSlot[i]->m_bySlotType)
	 {
  	   case DEV_DI_3DI477_6:
	   case DEV_DO_3DO760_6:
	   case DEV_PLC_CPU_260:
       case DEV_TCPCOM_IF_681:
            DestroyObject(CDgIOSlot,pT->m_pvSlot[i]->pChld);
	   break;
	   case DEV_AI_3AI375_6:
	   case DEV_AO_3AO775_6:
		    DestroyObject(CAnIOSlot,pT->m_pvSlot[i]->pChld);
	   break;
	   default:
	   break;
	 };
	}
	Delete(sizeof(CSlot*)*pT->m_pConfigTable->bySlotAmout,pT->m_pvSlot);
    DeleteObject(pT->m_pConfigTable);
}
DECLARE_SINGLE_CREATE(CComputer)
```
